Universal Robots URScript: azat_poduction_test_4.script

def azat_poduction_test_4():
  set_standard_analog_input_domain(0, 1)
  set_standard_analog_input_domain(1, 1)
  set_tool_analog_input_domain(0, 1)
  set_tool_analog_input_domain(1, 1)
  set_analog_outputdomain(0, 0)
  set_analog_outputdomain(1, 0)
  set_input_actions_to_default()
  set_target_payload(1.070000, [0.002000, 0.003000, 0.057000], [0.001723, 0.001723, 0.001723, 0.000000, 0.000000, 0.000000])
  set_tcp(p[0.0,0.0,0.0,0.0,0.0,0.0])
  set_gravity([0.0, 0.0, 9.82])
  set_tool_communication(True, 1000000, 2, 1, 1.5, 3.5)
  set_tool_output_mode(0)
  set_tool_digital_output_mode(0, 1)
  set_tool_digital_output_mode(1, 1)
  set_tool_voltage(0)
  set_safety_mode_transition_hardness(1)
  step_count_cf327c55_b5b8_495d_8ff7_12e031e14571 = 0.0
  thread Step_Counter_Thread_0ae96562_13f4_426a_a0a8_86ecd25231b4():
    while (True):
      step_count_cf327c55_b5b8_495d_8ff7_12e031e14571 = step_count_cf327c55_b5b8_495d_8ff7_12e031e14571 + 1.0
      sync()
    end
  end
  run Step_Counter_Thread_0ae96562_13f4_426a_a0a8_86ecd25231b4()
  global Plane_1=p[-0.700006141123905,1.3454883874109249E-6,0.3910559577028425,-1.2089868272251132,-1.2089999932245832,1.20858562628424]
  global Plane_2=p[0.0,0.0,0.0,0.0,0.0,0.0]
  global Point_1=p[0.6913645118948067,-0.12399382748223003,0.49223711947071,-1.2983729986843258,1.1259514972191385,-1.2203503861141718]
  $ 1 "Robot Program"
  $ 2 "Script: production_test_5.script"
  def Machining3():
    # Default parameters:
    global speed_ms = 0.3
    global speed_rads = 0.75
    global accel_mss = 3
    global accel_radss = 1.2
    global blend_radius_m = 0.001

    # Add subprograms here
    # Start of main program
    # Program generated by RoboDK v5.6.5 for UR10e on 16/10/2023 17:55:05
    # Using nominal kinematics.
    blend_radius_m = 0.001
    speed_ms = 1.000
    # set_reference(p[0.335000, -0.154000, 0.001500, 0.000000, 0.000000, 0.000000])
    set_tcp(p[0.000000, 0.000000, 0.252000, 0.000000, 0.000000, 0.000000])
    # Show Tool
    movej([0.158378, -1.225661, -2.546529, -0.940199, 1.570796, 1.729175],accel_radss,speed_rads,0,blend_radius_m)
    movel([0.158378, -1.324681, -2.603660, -0.784048, 1.570796, 1.729175],accel_mss,speed_ms,0,blend_radius_m)
    speed_ms = 0.003
    movel([0.158378, -1.328123, -2.605263, -0.779003, 1.570796, 1.729175],accel_mss,speed_ms,0,blend_radius_m)
    speed_ms = 0.008
    movel([0.158066, -1.328151, -2.605245, -0.778993, 1.570796, 1.728862],accel_mss,speed_ms,0,blend_radius_m)
    movel([0.148692, -1.330567, -2.603711, -0.778111, 1.570796, 1.719488],accel_mss,speed_ms,0,blend_radius_m)
    movel([0.142279, -1.332287, -2.602614, -0.777487, 1.570796, 1.713075],accel_mss,speed_ms,0,blend_radius_m)
    movel([0.124181, -1.337335, -2.599372, -0.775682, 1.570796, 1.694978],accel_mss,speed_ms,0,blend_radius_m)
    movel([0.122324, -1.350586, -2.590695, -0.771108, 1.570796, 1.693120],accel_mss,speed_ms,0,blend_radius_m)
    movel([0.141482, -1.345516, -2.594044, -0.772829, 1.570796, 1.712278],accel_mss,speed_ms,0,blend_radius_m)
    movel([0.146219, -1.344289, -2.594849, -0.773252, 1.570796, 1.717015],accel_mss,speed_ms,0,blend_radius_m)
    movel([0.150355, -1.343216, -2.595551, -0.773622, 1.570796, 1.721151],accel_mss,speed_ms,0,blend_radius_m)
    movel([0.155200, -1.341960, -2.596371, -0.774058, 1.570796, 1.725997],accel_mss,speed_ms,0,blend_radius_m)
    movel([0.155579, -1.341827, -2.596458, -0.774104, 1.570796, 1.726375],accel_mss,speed_ms,0,blend_radius_m)
    movel([0.156402, -1.341455, -2.596700, -0.774234, 1.570796, 1.727198],accel_mss,speed_ms,0,blend_radius_m)
    movel([0.157734, -1.333883, -2.601593, -0.776913, 1.570796, 1.728530],accel_mss,speed_ms,0,blend_radius_m)
    movel([0.158255, -1.330765, -2.603585, -0.778039, 1.570796, 1.729051],accel_mss,speed_ms,0,blend_radius_m)
    movel([0.158428, -1.329461, -2.604415, -0.778513, 1.570796, 1.729225],accel_mss,speed_ms,0,blend_radius_m)
    movel([0.158542, -1.328310, -2.605144, -0.778934, 1.570796, 1.729338],accel_mss,speed_ms,0,blend_radius_m)
    movel([0.158378, -1.328123, -2.605263, -0.779003, 1.570796, 1.729175],accel_mss,speed_ms,0,blend_radius_m)
    movel([0.158378, -1.331019, -2.606596, -0.774774, 1.570796, 1.729175],accel_mss,speed_ms,0,blend_radius_m)
    movel([0.158066, -1.331047, -2.606578, -0.774764, 1.570796, 1.728862],accel_mss,speed_ms,0,blend_radius_m)
    movel([0.148692, -1.333459, -2.605040, -0.773890, 1.570796, 1.719488],accel_mss,speed_ms,0,blend_radius_m)
    movel([0.142279, -1.335175, -2.603941, -0.773273, 1.570796, 1.713075],accel_mss,speed_ms,0,blend_radius_m)
    movel([0.124181, -1.340212, -2.600692, -0.771485, 1.570796, 1.694978],accel_mss,speed_ms,0,blend_radius_m)
    movel([0.122324, -1.353435, -2.591996, -0.766958, 1.570796, 1.693120],accel_mss,speed_ms,0,blend_radius_m)
    movel([0.141482, -1.348376, -2.595352, -0.768662, 1.570796, 1.712278],accel_mss,speed_ms,0,blend_radius_m)
    movel([0.146219, -1.347151, -2.596159, -0.769079, 1.570796, 1.717015],accel_mss,speed_ms,0,blend_radius_m)
    movel([0.150355, -1.346080, -2.596862, -0.769446, 1.570796, 1.721151],accel_mss,speed_ms,0,blend_radius_m)
    movel([0.155200, -1.344828, -2.597684, -0.769877, 1.570796, 1.725997],accel_mss,speed_ms,0,blend_radius_m)
    movel([0.155579, -1.344695, -2.597771, -0.769923, 1.570796, 1.726375],accel_mss,speed_ms,0,blend_radius_m)
    movel([0.156402, -1.344323, -2.598014, -0.770052, 1.570796, 1.727198],accel_mss,speed_ms,0,blend_radius_m)
    movel([0.157734, -1.336767, -2.602918, -0.772704, 1.570796, 1.728530],accel_mss,speed_ms,0,blend_radius_m)
    movel([0.158255, -1.333656, -2.604914, -0.773819, 1.570796, 1.729051],accel_mss,speed_ms,0,blend_radius_m)
    movel([0.158428, -1.332355, -2.605745, -0.774289, 1.570796, 1.729225],accel_mss,speed_ms,0,blend_radius_m)
    movel([0.158542, -1.331206, -2.606477, -0.774706, 1.570796, 1.729338],accel_mss,speed_ms,0,blend_radius_m)
    movel([0.158378, -1.331019, -2.606596, -0.774774, 1.570796, 1.729175],accel_mss,speed_ms,0,blend_radius_m)
    movel([0.158378, -1.297475, -2.590216, -0.824698, 1.570796, 1.729175],accel_mss,speed_ms,0,blend_radius_m)
    speed_ms = 1.000
    movel([0.162574, -1.288370, -2.595680, -0.828339, 1.570796, 1.733371],accel_mss,speed_ms,0,blend_radius_m)
    speed_ms = 0.008
    movel([0.162574, -1.315726, -2.609249, -0.787414, 1.570796, 1.733371],accel_mss,speed_ms,0,blend_radius_m)
    speed_ms = 0.003
    movel([0.162574, -1.319190, -2.610867, -0.782332, 1.570796, 1.733371],accel_mss,speed_ms,0,blend_radius_m)
    speed_ms = 0.008
    movel([0.162335, -1.318913, -2.611039, -0.782437, 1.570796, 1.733131],accel_mss,speed_ms,0,blend_radius_m)
    movel([0.162119, -1.318754, -2.611137, -0.782498, 1.570796, 1.732915],accel_mss,speed_ms,0,blend_radius_m)
    movel([0.161882, -1.318615, -2.611224, -0.782550, 1.570796, 1.732678],accel_mss,speed_ms,0,blend_radius_m)
    movel([0.161671, -1.318515, -2.611286, -0.782588, 1.570796, 1.732467],accel_mss,speed_ms,0,blend_radius_m)
    movel([0.161471, -1.318440, -2.611332, -0.782617, 1.570796, 1.732267],accel_mss,speed_ms,0,blend_radius_m)
    movel([0.160946, -1.318313, -2.611411, -0.782665, 1.570796, 1.731743],accel_mss,speed_ms,0,blend_radius_m)
    movel([0.160659, -1.318224, -2.611466, -0.782699, 1.570796, 1.731456],accel_mss,speed_ms,0,blend_radius_m)
    movel([0.160450, -1.318074, -2.611560, -0.782756, 1.570796, 1.731246],accel_mss,speed_ms,0,blend_radius_m)
    movel([0.160346, -1.317710, -2.611784, -0.782894, 1.570796, 1.731143],accel_mss,speed_ms,0,blend_radius_m)
    movel([0.160380, -1.317323, -2.612024, -0.783042, 1.570796, 1.731176],accel_mss,speed_ms,0,blend_radius_m)
    movel([0.160495, -1.316538, -2.612510, -0.783341, 1.570796, 1.731291],accel_mss,speed_ms,0,blend_radius_m)
    movel([0.160495, -1.316237, -2.612696, -0.783456, 1.570796, 1.731291],accel_mss,speed_ms,0,blend_radius_m)
    movel([0.160378, -1.316006, -2.612838, -0.783545, 1.570796, 1.731174],accel_mss,speed_ms,0,blend_radius_m)
    movel([0.160134, -1.315984, -2.612852, -0.783553, 1.570796, 1.730930],accel_mss,speed_ms,0,blend_radius_m)
    movel([0.159860, -1.316176, -2.612733, -0.783480, 1.570796, 1.730656],accel_mss,speed_ms,0,blend_radius_m)
    movel([0.159659, -1.316518, -2.612522, -0.783349, 1.570796, 1.730455],accel_mss,speed_ms,0,blend_radius_m)
    movel([0.159542, -1.316914, -2.612278, -0.783198, 1.570796, 1.730339],accel_mss,speed_ms,0,blend_radius_m)
    movel([0.159376, -1.317735, -2.611769, -0.782885, 1.570796, 1.730172],accel_mss,speed_ms,0,blend_radius_m)
    movel([0.159287, -1.318121, -2.611530, -0.782738, 1.570796, 1.730084],accel_mss,speed_ms,0,blend_radius_m)
    movel([0.159193, -1.318381, -2.611369, -0.782639, 1.570796, 1.729989],accel_mss,speed_ms,0,blend_radius_m)
    movel([0.158977, -1.318693, -2.611175, -0.782521, 1.570796, 1.729773],accel_mss,speed_ms,0,blend_radius_m)
    movel([0.158624, -1.318877, -2.611061, -0.782451, 1.570796, 1.729420],accel_mss,speed_ms,0,blend_radius_m)
    movel([0.158228, -1.319117, -2.610912, -0.782360, 1.570796, 1.729024],accel_mss,speed_ms,0,blend_radius_m)
    movel([0.157857, -1.319400, -2.610736, -0.782253, 1.570796, 1.728653],accel_mss,speed_ms,0,blend_radius_m)
    movel([0.157491, -1.319715, -2.610541, -0.782134, 1.570796, 1.728288],accel_mss,speed_ms,0,blend_radius_m)
    movel([0.157078, -1.320110, -2.610294, -0.781984, 1.570796, 1.727875],accel_mss,speed_ms,0,blend_radius_m)
    movel([0.156693, -1.320526, -2.610035, -0.781828, 1.570796, 1.727489],accel_mss,speed_ms,0,blend_radius_m)
    movel([0.156421, -1.320857, -2.609829, -0.781703, 1.570796, 1.727218],accel_mss,speed_ms,0,blend_radius_m)
    movel([0.156220, -1.321169, -2.609634, -0.781585, 1.570796, 1.727016],accel_mss,speed_ms,0,blend_radius_m)
    movel([0.156088, -1.321431, -2.609471, -0.781487, 1.570796, 1.726884],accel_mss,speed_ms,0,blend_radius_m)
    movel([0.155989, -1.321691, -2.609309, -0.781390, 1.570796, 1.726785],accel_mss,speed_ms,0,blend_radius_m)
    movel([0.155886, -1.322078, -2.609067, -0.781244, 1.570796, 1.726682],accel_mss,speed_ms,0,blend_radius_m)
    movel([0.155804, -1.322477, -2.608817, -0.781095, 1.570796, 1.726600],accel_mss,speed_ms,0,blend_radius_m)
    movel([0.155743, -1.322882, -2.608563, -0.780943, 1.570796, 1.726540],accel_mss,speed_ms,0,blend_radius_m)
    movel([0.155711, -1.323271, -2.608320, -0.780798, 1.570796, 1.726508],accel_mss,speed_ms,0,blend_radius_m)
    movel([0.155722, -1.323501, -2.608176, -0.780712, 1.570796, 1.726518],accel_mss,speed_ms,0,blend_radius_m)
    movel([0.155763, -1.323714, -2.608042, -0.780633, 1.570796, 1.726560],accel_mss,speed_ms,0,blend_radius_m)
    movel([0.155867, -1.323948, -2.607895, -0.780546, 1.570796, 1.726664],accel_mss,speed_ms,0,blend_radius_m)
    movel([0.156031, -1.324157, -2.607764, -0.780468, 1.570796, 1.726827],accel_mss,speed_ms,0,blend_radius_m)
    movel([0.156304, -1.324405, -2.607608, -0.780376, 1.570796, 1.727100],accel_mss,speed_ms,0,blend_radius_m)
    movel([0.156613, -1.324619, -2.607474, -0.780296, 1.570796, 1.727410],accel_mss,speed_ms,0,blend_radius_m)
    movel([0.156897, -1.324765, -2.607382, -0.780242, 1.570796, 1.727693],accel_mss,speed_ms,0,blend_radius_m)
    movel([0.157199, -1.324874, -2.607314, -0.780202, 1.570796, 1.727995],accel_mss,speed_ms,0,blend_radius_m)
    movel([0.157457, -1.324930, -2.607278, -0.780181, 1.570796, 1.728254],accel_mss,speed_ms,0,blend_radius_m)
    movel([0.157789, -1.324899, -2.607298, -0.780192, 1.570796, 1.728585],accel_mss,speed_ms,0,blend_radius_m)
    movel([0.157974, -1.325070, -2.607190, -0.780129, 1.570796, 1.728770],accel_mss,speed_ms,0,blend_radius_m)
    movel([0.158001, -1.325401, -2.606982, -0.780006, 1.570796, 1.728798],accel_mss,speed_ms,0,blend_radius_m)
    movel([0.157952, -1.325794, -2.606734, -0.779861, 1.570796, 1.728748],accel_mss,speed_ms,0,blend_radius_m)
    movel([0.157831, -1.326555, -2.606254, -0.779580, 1.570796, 1.728627],accel_mss,speed_ms,0,blend_radius_m)
    movel([0.157799, -1.326893, -2.606041, -0.779455, 1.570796, 1.728595],accel_mss,speed_ms,0,blend_radius_m)
    movel([0.157855, -1.327134, -2.605889, -0.779366, 1.570796, 1.728651],accel_mss,speed_ms,0,blend_radius_m)
    movel([0.158126, -1.327223, -2.605832, -0.779333, 1.570796, 1.728923],accel_mss,speed_ms,0,blend_radius_m)
    movel([0.158515, -1.327123, -2.605896, -0.779370, 1.570796, 1.729311],accel_mss,speed_ms,0,blend_radius_m)
    movel([0.158817, -1.326911, -2.606030, -0.779448, 1.570796, 1.729614],accel_mss,speed_ms,0,blend_radius_m)
    movel([0.158967, -1.326652, -2.606193, -0.779544, 1.570796, 1.729763],accel_mss,speed_ms,0,blend_radius_m)
    movel([0.159238, -1.325438, -2.606959, -0.779993, 1.570796, 1.730035],accel_mss,speed_ms,0,blend_radius_m)
    movel([0.159346, -1.325001, -2.607234, -0.780154, 1.570796, 1.730143],accel_mss,speed_ms,0,blend_radius_m)
    movel([0.159523, -1.324631, -2.607466, -0.780292, 1.570796, 1.730320],accel_mss,speed_ms,0,blend_radius_m)
    movel([0.159843, -1.324297, -2.607676, -0.780416, 1.570796, 1.730640],accel_mss,speed_ms,0,blend_radius_m)
    movel([0.160113, -1.324104, -2.607797, -0.780487, 1.570796, 1.730909],accel_mss,speed_ms,0,blend_radius_m)
    movel([0.160523, -1.323848, -2.607958, -0.780583, 1.570796, 1.731320],accel_mss,speed_ms,0,blend_radius_m)
    movel([0.161031, -1.323475, -2.608192, -0.780722, 1.570796, 1.731827],accel_mss,speed_ms,0,blend_radius_m)
    movel([0.161287, -1.323244, -2.608337, -0.780808, 1.570796, 1.732084],accel_mss,speed_ms,0,blend_radius_m)
    movel([0.161561, -1.322963, -2.608513, -0.780913, 1.570796, 1.732357],accel_mss,speed_ms,0,blend_radius_m)
    movel([0.161831, -1.322642, -2.608714, -0.781033, 1.570796, 1.732628],accel_mss,speed_ms,0,blend_radius_m)
    movel([0.162070, -1.322314, -2.608919, -0.781156, 1.570796, 1.732867],accel_mss,speed_ms,0,blend_radius_m)
    movel([0.162281, -1.321976, -2.609131, -0.781283, 1.570796, 1.733077],accel_mss,speed_ms,0,blend_radius_m)
    movel([0.162481, -1.321587, -2.609373, -0.781428, 1.570796, 1.733277],accel_mss,speed_ms,0,blend_radius_m)
    movel([0.162638, -1.321193, -2.609619, -0.781576, 1.570796, 1.733434],accel_mss,speed_ms,0,blend_radius_m)
    movel([0.162748, -1.320809, -2.609859, -0.781721, 1.570796, 1.733545],accel_mss,speed_ms,0,blend_radius_m)
    movel([0.162812, -1.320429, -2.610096, -0.781864, 1.570796, 1.733608],accel_mss,speed_ms,0,blend_radius_m)
    movel([0.162827, -1.320082, -2.610312, -0.781995, 1.570796, 1.733623],accel_mss,speed_ms,0,blend_radius_m)
    movel([0.162792, -1.319758, -2.610514, -0.782118, 1.570796, 1.733588],accel_mss,speed_ms,0,blend_radius_m)
    movel([0.162706, -1.319460, -2.610699, -0.782230, 1.570796, 1.733502],accel_mss,speed_ms,0,blend_radius_m)
    movel([0.162574, -1.319190, -2.610867, -0.782332, 1.570796, 1.733371],accel_mss,speed_ms,0,blend_radius_m)
    movel([0.162574, -1.322104, -2.612212, -0.778073, 1.570796, 1.733371],accel_mss,speed_ms,0,blend_radius_m)
    movel([0.162335, -1.321828, -2.612385, -0.778177, 1.570796, 1.733131],accel_mss,speed_ms,0,blend_radius_m)
    movel([0.162119, -1.321670, -2.612483, -0.778236, 1.570796, 1.732915],accel_mss,speed_ms,0,blend_radius_m)
    movel([0.161882, -1.321531, -2.612570, -0.778289, 1.570796, 1.732678],accel_mss,speed_ms,0,blend_radius_m)
    movel([0.161671, -1.321431, -2.612632, -0.778326, 1.570796, 1.732467],accel_mss,speed_ms,0,blend_radius_m)
    movel([0.161471, -1.321356, -2.612679, -0.778354, 1.570796, 1.732267],accel_mss,speed_ms,0,blend_radius_m)
    movel([0.160946, -1.321230, -2.612757, -0.778402, 1.570796, 1.731743],accel_mss,speed_ms,0,blend_radius_m)
    movel([0.160659, -1.321141, -2.612813, -0.778436, 1.570796, 1.731456],accel_mss,speed_ms,0,blend_radius_m)
    movel([0.160450, -1.320990, -2.612906, -0.778492, 1.570796, 1.731246],accel_mss,speed_ms,0,blend_radius_m)
    movel([0.160346, -1.320628, -2.613132, -0.778629, 1.570796, 1.731143],accel_mss,speed_ms,0,blend_radius_m)
    movel([0.160380, -1.320241, -2.613372, -0.778775, 1.570796, 1.731176],accel_mss,speed_ms,0,blend_radius_m)
    movel([0.160495, -1.319457, -2.613859, -0.779072, 1.570796, 1.731291],accel_mss,speed_ms,0,blend_radius_m)
    movel([0.160495, -1.319157, -2.614045, -0.779186, 1.570796, 1.731291],accel_mss,speed_ms,0,blend_radius_m)
    movel([0.160378, -1.318927, -2.614188, -0.779274, 1.570796, 1.731174],accel_mss,speed_ms,0,blend_radius_m)
    movel([0.160134, -1.318905, -2.614201, -0.779282, 1.570796, 1.730930],accel_mss,speed_ms,0,blend_radius_m)
    movel([0.159860, -1.319097, -2.614083, -0.779209, 1.570796, 1.730656],accel_mss,speed_ms,0,blend_radius_m)
    movel([0.159659, -1.319438, -2.613871, -0.779080, 1.570796, 1.730455],accel_mss,speed_ms,0,blend_radius_m)
    movel([0.159542, -1.319833, -2.613626, -0.778930, 1.570796, 1.730339],accel_mss,speed_ms,0,blend_radius_m)
    movel([0.159376, -1.320653, -2.613116, -0.778620, 1.570796, 1.730172],accel_mss,speed_ms,0,blend_radius_m)
    movel([0.159287, -1.321037, -2.612877, -0.778475, 1.570796, 1.730084],accel_mss,speed_ms,0,blend_radius_m)
    movel([0.159193, -1.321297, -2.612716, -0.778377, 1.570796, 1.729989],accel_mss,speed_ms,0,blend_radius_m)
    movel([0.158977, -1.321608, -2.612521, -0.778259, 1.570796, 1.729773],accel_mss,speed_ms,0,blend_radius_m)
    movel([0.158624, -1.321792, -2.612407, -0.778190, 1.570796, 1.729420],accel_mss,speed_ms,0,blend_radius_m)
    movel([0.158228, -1.322031, -2.612258, -0.778100, 1.570796, 1.729024],accel_mss,speed_ms,0,blend_radius_m)
    movel([0.157857, -1.322314, -2.612081, -0.777994, 1.570796, 1.728653],accel_mss,speed_ms,0,blend_radius_m)
    movel([0.157491, -1.322628, -2.611885, -0.777876, 1.570796, 1.728288],accel_mss,speed_ms,0,blend_radius_m)
    movel([0.157078, -1.323023, -2.611638, -0.777728, 1.570796, 1.727875],accel_mss,speed_ms,0,blend_radius_m)
    movel([0.156693, -1.323438, -2.611379, -0.777572, 1.570796, 1.727489],accel_mss,speed_ms,0,blend_radius_m)
    movel([0.156421, -1.323768, -2.611172, -0.777449, 1.570796, 1.727218],accel_mss,speed_ms,0,blend_radius_m)
    movel([0.156220, -1.324080, -2.610977, -0.777332, 1.570796, 1.727016],accel_mss,speed_ms,0,blend_radius_m)
    movel([0.156088, -1.324341, -2.610813, -0.777235, 1.570796, 1.726884],accel_mss,speed_ms,0,blend_radius_m)
    movel([0.155989, -1.324600, -2.610650, -0.777138, 1.570796, 1.726785],accel_mss,speed_ms,0,blend_radius_m)
    movel([0.155886, -1.324986, -2.610408, -0.776994, 1.570796, 1.726682],accel_mss,speed_ms,0,blend_radius_m)
    movel([0.155804, -1.325385, -2.610158, -0.776846, 1.570796, 1.726600],accel_mss,speed_ms,0,blend_radius_m)
    movel([0.155743, -1.325789, -2.609903, -0.776696, 1.570796, 1.726540],accel_mss,speed_ms,0,blend_radius_m)
    movel([0.155711, -1.326177, -2.609660, -0.776552, 1.570796, 1.726508],accel_mss,speed_ms,0,blend_radius_m)
    movel([0.155722, -1.326407, -2.609515, -0.776467, 1.570796, 1.726518],accel_mss,speed_ms,0,blend_radius_m)
    movel([0.155763, -1.326620, -2.609381, -0.776388, 1.570796, 1.726560],accel_mss,speed_ms,0,blend_radius_m)
    movel([0.155867, -1.326853, -2.609234, -0.776302, 1.570796, 1.726664],accel_mss,speed_ms,0,blend_radius_m)
    movel([0.156031, -1.327061, -2.609103, -0.776225, 1.570796, 1.726827],accel_mss,speed_ms,0,blend_radius_m)
    movel([0.156304, -1.327309, -2.608946, -0.776134, 1.570796, 1.727100],accel_mss,speed_ms,0,blend_radius_m)
    movel([0.156613, -1.327523, -2.608811, -0.776055, 1.570796, 1.727410],accel_mss,speed_ms,0,blend_radius_m)
    movel([0.156897, -1.327668, -2.608719, -0.776001, 1.570796, 1.727693],accel_mss,speed_ms,0,blend_radius_m)
    movel([0.157199, -1.327777, -2.608651, -0.775961, 1.570796, 1.727995],accel_mss,speed_ms,0,blend_radius_m)
    movel([0.157457, -1.327833, -2.608615, -0.775941, 1.570796, 1.728254],accel_mss,speed_ms,0,blend_radius_m)
    movel([0.157789, -1.327802, -2.608635, -0.775952, 1.570796, 1.728585],accel_mss,speed_ms,0,blend_radius_m)
    movel([0.157974, -1.327973, -2.608527, -0.775889, 1.570796, 1.728770],accel_mss,speed_ms,0,blend_radius_m)
    movel([0.158001, -1.328303, -2.608319, -0.775768, 1.570796, 1.728798],accel_mss,speed_ms,0,blend_radius_m)
    movel([0.157952, -1.328695, -2.608070, -0.775623, 1.570796, 1.728748],accel_mss,speed_ms,0,blend_radius_m)
    movel([0.157831, -1.329455, -2.607589, -0.775345, 1.570796, 1.728627],accel_mss,speed_ms,0,blend_radius_m)
    movel([0.157799, -1.329792, -2.607375, -0.775222, 1.570796, 1.728595],accel_mss,speed_ms,0,blend_radius_m)
    movel([0.157855, -1.330032, -2.607223, -0.775134, 1.570796, 1.728651],accel_mss,speed_ms,0,blend_radius_m)
    movel([0.158126, -1.330121, -2.607166, -0.775101, 1.570796, 1.728923],accel_mss,speed_ms,0,blend_radius_m)
    movel([0.158515, -1.330022, -2.607230, -0.775138, 1.570796, 1.729311],accel_mss,speed_ms,0,blend_radius_m)
    movel([0.158817, -1.329810, -2.607364, -0.775215, 1.570796, 1.729614],accel_mss,speed_ms,0,blend_radius_m)
    movel([0.158967, -1.329551, -2.607528, -0.775310, 1.570796, 1.729763],accel_mss,speed_ms,0,blend_radius_m)
    movel([0.159238, -1.328339, -2.608295, -0.775754, 1.570796, 1.730035],accel_mss,speed_ms,0,blend_radius_m)
    movel([0.159346, -1.327904, -2.608571, -0.775915, 1.570796, 1.730143],accel_mss,speed_ms,0,blend_radius_m)
    movel([0.159523, -1.327535, -2.608804, -0.776051, 1.570796, 1.730320],accel_mss,speed_ms,0,blend_radius_m)
    movel([0.159843, -1.327202, -2.609014, -0.776173, 1.570796, 1.730640],accel_mss,speed_ms,0,blend_radius_m)
    movel([0.160113, -1.327009, -2.609135, -0.776245, 1.570796, 1.730909],accel_mss,speed_ms,0,blend_radius_m)
    movel([0.160523, -1.326753, -2.609297, -0.776339, 1.570796, 1.731320],accel_mss,speed_ms,0,blend_radius_m)
    movel([0.161031, -1.326381, -2.609531, -0.776477, 1.570796, 1.731827],accel_mss,speed_ms,0,blend_radius_m)
    movel([0.161287, -1.326150, -2.609676, -0.776562, 1.570796, 1.732084],accel_mss,speed_ms,0,blend_radius_m)
    movel([0.161561, -1.325870, -2.609853, -0.776666, 1.570796, 1.732357],accel_mss,speed_ms,0,blend_radius_m)
    movel([0.161831, -1.325549, -2.610054, -0.776785, 1.570796, 1.732628],accel_mss,speed_ms,0,blend_radius_m)
    movel([0.162070, -1.325223, -2.610260, -0.776907, 1.570796, 1.732867],accel_mss,speed_ms,0,blend_radius_m)
    movel([0.162281, -1.324885, -2.610472, -0.777032, 1.570796, 1.733077],accel_mss,speed_ms,0,blend_radius_m)
    movel([0.162481, -1.324497, -2.610715, -0.777177, 1.570796, 1.733277],accel_mss,speed_ms,0,blend_radius_m)
    movel([0.162638, -1.324104, -2.610962, -0.777324, 1.570796, 1.733434],accel_mss,speed_ms,0,blend_radius_m)
    movel([0.162748, -1.323720, -2.611202, -0.777467, 1.570796, 1.733545],accel_mss,speed_ms,0,blend_radius_m)
    movel([0.162812, -1.323341, -2.611439, -0.777609, 1.570796, 1.733608],accel_mss,speed_ms,0,blend_radius_m)
    movel([0.162827, -1.322995, -2.611656, -0.777738, 1.570796, 1.733623],accel_mss,speed_ms,0,blend_radius_m)
    movel([0.162792, -1.322671, -2.611858, -0.777860, 1.570796, 1.733588],accel_mss,speed_ms,0,blend_radius_m)
    movel([0.162706, -1.322374, -2.612044, -0.777971, 1.570796, 1.733502],accel_mss,speed_ms,0,blend_radius_m)
    movel([0.162574, -1.322104, -2.612212, -0.778073, 1.570796, 1.733371],accel_mss,speed_ms,0,blend_radius_m)
    movel([0.162574, -1.288370, -2.595680, -0.828339, 1.570796, 1.733371],accel_mss,speed_ms,0,blend_radius_m)
    speed_ms = 1.000
    movel([0.151112, -1.291543, -2.593788, -0.827058, 1.570796, 1.721909],accel_mss,speed_ms,0,blend_radius_m)
    speed_ms = 0.008
    movel([0.151112, -1.318847, -2.607313, -0.786229, 1.570796, 1.721909],accel_mss,speed_ms,0,blend_radius_m)
    speed_ms = 0.003
    movel([0.151112, -1.322303, -2.608926, -0.781160, 1.570796, 1.721909],accel_mss,speed_ms,0,blend_radius_m)
    speed_ms = 0.008
    movel([0.151013, -1.322091, -2.609058, -0.781239, 1.570796, 1.721810],accel_mss,speed_ms,0,blend_radius_m)
    movel([0.150875, -1.321902, -2.609177, -0.781310, 1.570796, 1.721672],accel_mss,speed_ms,0,blend_radius_m)
    movel([0.150690, -1.321720, -2.609291, -0.781379, 1.570796, 1.721486],accel_mss,speed_ms,0,blend_radius_m)
    movel([0.150469, -1.321563, -2.609388, -0.781437, 1.570796, 1.721266],accel_mss,speed_ms,0,blend_radius_m)
    movel([0.150261, -1.321456, -2.609455, -0.781478, 1.570796, 1.721057],accel_mss,speed_ms,0,blend_radius_m)
    movel([0.150043, -1.321372, -2.609508, -0.781509, 1.570796, 1.720840],accel_mss,speed_ms,0,blend_radius_m)
    movel([0.149464, -1.321243, -2.609588, -0.781558, 1.570796, 1.720261],accel_mss,speed_ms,0,blend_radius_m)
    movel([0.149161, -1.321155, -2.609643, -0.781591, 1.570796, 1.719957],accel_mss,speed_ms,0,blend_radius_m)
    movel([0.148935, -1.320995, -2.609743, -0.781651, 1.570796, 1.719732],accel_mss,speed_ms,0,blend_radius_m)
    movel([0.148830, -1.320661, -2.609951, -0.781777, 1.570796, 1.719627],accel_mss,speed_ms,0,blend_radius_m)
    movel([0.148858, -1.320296, -2.610179, -0.781914, 1.570796, 1.719654],accel_mss,speed_ms,0,blend_radius_m)
    movel([0.148950, -1.319577, -2.610626, -0.782186, 1.570796, 1.719746],accel_mss,speed_ms,0,blend_radius_m)
    movel([0.148946, -1.319296, -2.610801, -0.782292, 1.570796, 1.719742],accel_mss,speed_ms,0,blend_radius_m)
    movel([0.148829, -1.319077, -2.610937, -0.782375, 1.570796, 1.719625],accel_mss,speed_ms,0,blend_radius_m)
    movel([0.148588, -1.319055, -2.610951, -0.782384, 1.570796, 1.719384],accel_mss,speed_ms,0,blend_radius_m)
    movel([0.148325, -1.319220, -2.610848, -0.782321, 1.570796, 1.719122],accel_mss,speed_ms,0,blend_radius_m)
    movel([0.148131, -1.319516, -2.610664, -0.782209, 1.570796, 1.718927],accel_mss,speed_ms,0,blend_radius_m)
    movel([0.148031, -1.319812, -2.610480, -0.782097, 1.570796, 1.718827],accel_mss,speed_ms,0,blend_radius_m)
    movel([0.147884, -1.320528, -2.610034, -0.781827, 1.570796, 1.718680],accel_mss,speed_ms,0,blend_radius_m)
    movel([0.147783, -1.320906, -2.609798, -0.781684, 1.570796, 1.718580],accel_mss,speed_ms,0,blend_radius_m)
    movel([0.147549, -1.321339, -2.609529, -0.781522, 1.570796, 1.718345],accel_mss,speed_ms,0,blend_radius_m)
    movel([0.147223, -1.321676, -2.609318, -0.781395, 1.570796, 1.718019],accel_mss,speed_ms,0,blend_radius_m)
    movel([0.146841, -1.321972, -2.609133, -0.781284, 1.570796, 1.717637],accel_mss,speed_ms,0,blend_radius_m)
    movel([0.146144, -1.322480, -2.608815, -0.781094, 1.570796, 1.716940],accel_mss,speed_ms,0,blend_radius_m)
    movel([0.145876, -1.322704, -2.608675, -0.781010, 1.570796, 1.716672],accel_mss,speed_ms,0,blend_radius_m)
    movel([0.145621, -1.322940, -2.608528, -0.780922, 1.570796, 1.716417],accel_mss,speed_ms,0,blend_radius_m)
    movel([0.145339, -1.323235, -2.608342, -0.780811, 1.570796, 1.716135],accel_mss,speed_ms,0,blend_radius_m)
    movel([0.145080, -1.323543, -2.608150, -0.780697, 1.570796, 1.715876],accel_mss,speed_ms,0,blend_radius_m)
    movel([0.144848, -1.323861, -2.607950, -0.780578, 1.570796, 1.715644],accel_mss,speed_ms,0,blend_radius_m)
    movel([0.144646, -1.324183, -2.607748, -0.780458, 1.570796, 1.715442],accel_mss,speed_ms,0,blend_radius_m)
    movel([0.144474, -1.324508, -2.607544, -0.780337, 1.570796, 1.715270],accel_mss,speed_ms,0,blend_radius_m)
    movel([0.144335, -1.324833, -2.607340, -0.780217, 1.570796, 1.715131],accel_mss,speed_ms,0,blend_radius_m)
    movel([0.144229, -1.325155, -2.607137, -0.780097, 1.570796, 1.715025],accel_mss,speed_ms,0,blend_radius_m)
    movel([0.144155, -1.325473, -2.606936, -0.779979, 1.570796, 1.714951],accel_mss,speed_ms,0,blend_radius_m)
    movel([0.144121, -1.325776, -2.606746, -0.779867, 1.570796, 1.714917],accel_mss,speed_ms,0,blend_radius_m)
    movel([0.144119, -1.326068, -2.606562, -0.779759, 1.570796, 1.714916],accel_mss,speed_ms,0,blend_radius_m)
    movel([0.144153, -1.326345, -2.606387, -0.779657, 1.570796, 1.714949],accel_mss,speed_ms,0,blend_radius_m)
    movel([0.144225, -1.326603, -2.606224, -0.779562, 1.570796, 1.715022],accel_mss,speed_ms,0,blend_radius_m)
    movel([0.144335, -1.326851, -2.606068, -0.779471, 1.570796, 1.715131],accel_mss,speed_ms,0,blend_radius_m)
    movel([0.144483, -1.327074, -2.605926, -0.779388, 1.570796, 1.715280],accel_mss,speed_ms,0,blend_radius_m)
    movel([0.144667, -1.327270, -2.605803, -0.779316, 1.570796, 1.715463],accel_mss,speed_ms,0,blend_radius_m)
    movel([0.144884, -1.327432, -2.605700, -0.779257, 1.570796, 1.715680],accel_mss,speed_ms,0,blend_radius_m)
    movel([0.145095, -1.327550, -2.605626, -0.779213, 1.570796, 1.715891],accel_mss,speed_ms,0,blend_radius_m)
    movel([0.145328, -1.327640, -2.605569, -0.779180, 1.570796, 1.716125],accel_mss,speed_ms,0,blend_radius_m)
    movel([0.145936, -1.327776, -2.605482, -0.779130, 1.570796, 1.716732],accel_mss,speed_ms,0,blend_radius_m)
    movel([0.146236, -1.327862, -2.605428, -0.779099, 1.570796, 1.717032],accel_mss,speed_ms,0,blend_radius_m)
    movel([0.146465, -1.328034, -2.605319, -0.779035, 1.570796, 1.717262],accel_mss,speed_ms,0,blend_radius_m)
    movel([0.146559, -1.328359, -2.605114, -0.778916, 1.570796, 1.717355],accel_mss,speed_ms,0,blend_radius_m)
    movel([0.146535, -1.328716, -2.604887, -0.778785, 1.570796, 1.717332],accel_mss,speed_ms,0,blend_radius_m)
    movel([0.146450, -1.329360, -2.604479, -0.778550, 1.570796, 1.717246],accel_mss,speed_ms,0,blend_radius_m)
    movel([0.146442, -1.329634, -2.604305, -0.778450, 1.570796, 1.717239],accel_mss,speed_ms,0,blend_radius_m)
    movel([0.146505, -1.329850, -2.604167, -0.778371, 1.570796, 1.717302],accel_mss,speed_ms,0,blend_radius_m)
    movel([0.146734, -1.329948, -2.604105, -0.778336, 1.570796, 1.717530],accel_mss,speed_ms,0,blend_radius_m)
    movel([0.147042, -1.329791, -2.604205, -0.778393, 1.570796, 1.717839],accel_mss,speed_ms,0,blend_radius_m)
    movel([0.147221, -1.329551, -2.604357, -0.778480, 1.570796, 1.718017],accel_mss,speed_ms,0,blend_radius_m)
    movel([0.147341, -1.329239, -2.604556, -0.778595, 1.570796, 1.718137],accel_mss,speed_ms,0,blend_radius_m)
    movel([0.147409, -1.328946, -2.604741, -0.778701, 1.570796, 1.718206],accel_mss,speed_ms,0,blend_radius_m)
    movel([0.147506, -1.328440, -2.605062, -0.778887, 1.570796, 1.718302],accel_mss,speed_ms,0,blend_radius_m)
    movel([0.147604, -1.328062, -2.605302, -0.779025, 1.570796, 1.718400],accel_mss,speed_ms,0,blend_radius_m)
    movel([0.147844, -1.327635, -2.605572, -0.779182, 1.570796, 1.718640],accel_mss,speed_ms,0,blend_radius_m)
    movel([0.148134, -1.327351, -2.605751, -0.779286, 1.570796, 1.718930],accel_mss,speed_ms,0,blend_radius_m)
    movel([0.148494, -1.327087, -2.605918, -0.779383, 1.570796, 1.719290],accel_mss,speed_ms,0,blend_radius_m)
    movel([0.149174, -1.326623, -2.606212, -0.779555, 1.570796, 1.719970],accel_mss,speed_ms,0,blend_radius_m)
    movel([0.149442, -1.326410, -2.606346, -0.779633, 1.570796, 1.720239],accel_mss,speed_ms,0,blend_radius_m)
    movel([0.149695, -1.326189, -2.606486, -0.779715, 1.570796, 1.720491],accel_mss,speed_ms,0,blend_radius_m)
    movel([0.149972, -1.325910, -2.606661, -0.779818, 1.570796, 1.720768],accel_mss,speed_ms,0,blend_radius_m)
    movel([0.150223, -1.325623, -2.606842, -0.779924, 1.570796, 1.721019],accel_mss,speed_ms,0,blend_radius_m)
    movel([0.150448, -1.325324, -2.607031, -0.780035, 1.570796, 1.721244],accel_mss,speed_ms,0,blend_radius_m)
    movel([0.150644, -1.325016, -2.607224, -0.780149, 1.570796, 1.721440],accel_mss,speed_ms,0,blend_radius_m)
    movel([0.150915, -1.324520, -2.607536, -0.780333, 1.570796, 1.721712],accel_mss,speed_ms,0,blend_radius_m)
    movel([0.151162, -1.324023, -2.607848, -0.780518, 1.570796, 1.721958],accel_mss,speed_ms,0,blend_radius_m)
    movel([0.151258, -1.323772, -2.608006, -0.780611, 1.570796, 1.722054],accel_mss,speed_ms,0,blend_radius_m)
    movel([0.151320, -1.323525, -2.608161, -0.780703, 1.570796, 1.722116],accel_mss,speed_ms,0,blend_radius_m)
    movel([0.151343, -1.323285, -2.608311, -0.780793, 1.570796, 1.722139],accel_mss,speed_ms,0,blend_radius_m)
    movel([0.151325, -1.323059, -2.608453, -0.780877, 1.570796, 1.722121],accel_mss,speed_ms,0,blend_radius_m)
    movel([0.151234, -1.322683, -2.608688, -0.781018, 1.570796, 1.722030],accel_mss,speed_ms,0,blend_radius_m)
    movel([0.151112, -1.322303, -2.608926, -0.781160, 1.570796, 1.721909],accel_mss,speed_ms,0,blend_radius_m)
    movel([0.151112, -1.325211, -2.610267, -0.776911, 1.570796, 1.721909],accel_mss,speed_ms,0,blend_radius_m)
    movel([0.151013, -1.325000, -2.610399, -0.776989, 1.570796, 1.721810],accel_mss,speed_ms,0,blend_radius_m)
    movel([0.150875, -1.324811, -2.610518, -0.777060, 1.570796, 1.721672],accel_mss,speed_ms,0,blend_radius_m)
    movel([0.150690, -1.324629, -2.610632, -0.777128, 1.570796, 1.721486],accel_mss,speed_ms,0,blend_radius_m)
    movel([0.150469, -1.324473, -2.610730, -0.777186, 1.570796, 1.721266],accel_mss,speed_ms,0,blend_radius_m)
    movel([0.150261, -1.324366, -2.610797, -0.777226, 1.570796, 1.721057],accel_mss,speed_ms,0,blend_radius_m)
    movel([0.150043, -1.324282, -2.610850, -0.777257, 1.570796, 1.720840],accel_mss,speed_ms,0,blend_radius_m)
    movel([0.149464, -1.324153, -2.610931, -0.777305, 1.570796, 1.720261],accel_mss,speed_ms,0,blend_radius_m)
    movel([0.149161, -1.324065, -2.610986, -0.777338, 1.570796, 1.719957],accel_mss,speed_ms,0,blend_radius_m)
    movel([0.148935, -1.323906, -2.611086, -0.777397, 1.570796, 1.719732],accel_mss,speed_ms,0,blend_radius_m)
    movel([0.148830, -1.323573, -2.611294, -0.777522, 1.570796, 1.719627],accel_mss,speed_ms,0,blend_radius_m)
    movel([0.148858, -1.323208, -2.611523, -0.777658, 1.570796, 1.719654],accel_mss,speed_ms,0,blend_radius_m)
    movel([0.148950, -1.322491, -2.611971, -0.777927, 1.570796, 1.719746],accel_mss,speed_ms,0,blend_radius_m)
    movel([0.148946, -1.322210, -2.612146, -0.778033, 1.570796, 1.719742],accel_mss,speed_ms,0,blend_radius_m)
    movel([0.148829, -1.321992, -2.612282, -0.778115, 1.570796, 1.719625],accel_mss,speed_ms,0,blend_radius_m)
    movel([0.148588, -1.321969, -2.612296, -0.778123, 1.570796, 1.719384],accel_mss,speed_ms,0,blend_radius_m)
    movel([0.148325, -1.322134, -2.612193, -0.778061, 1.570796, 1.719122],accel_mss,speed_ms,0,blend_radius_m)
    movel([0.148131, -1.322430, -2.612009, -0.777950, 1.570796, 1.718927],accel_mss,speed_ms,0,blend_radius_m)
    movel([0.148031, -1.322725, -2.611825, -0.777840, 1.570796, 1.718827],accel_mss,speed_ms,0,blend_radius_m)
    movel([0.147884, -1.323440, -2.611377, -0.777572, 1.570796, 1.718680],accel_mss,speed_ms,0,blend_radius_m)
    movel([0.147783, -1.323818, -2.611141, -0.777430, 1.570796, 1.718580],accel_mss,speed_ms,0,blend_radius_m)
    movel([0.147549, -1.324249, -2.610871, -0.777269, 1.570796, 1.718345],accel_mss,speed_ms,0,blend_radius_m)
    movel([0.147223, -1.324586, -2.610660, -0.777144, 1.570796, 1.718019],accel_mss,speed_ms,0,blend_radius_m)
    movel([0.146841, -1.324881, -2.610474, -0.777034, 1.570796, 1.717637],accel_mss,speed_ms,0,blend_radius_m)
    movel([0.146144, -1.325388, -2.610156, -0.776845, 1.570796, 1.716940],accel_mss,speed_ms,0,blend_radius_m)
    movel([0.145876, -1.325611, -2.610016, -0.776762, 1.570796, 1.716672],accel_mss,speed_ms,0,blend_radius_m)
    movel([0.145621, -1.325846, -2.609868, -0.776675, 1.570796, 1.716417],accel_mss,speed_ms,0,blend_radius_m)
    movel([0.145339, -1.326142, -2.609682, -0.776566, 1.570796, 1.716135],accel_mss,speed_ms,0,blend_radius_m)
    movel([0.145080, -1.326448, -2.609489, -0.776452, 1.570796, 1.715876],accel_mss,speed_ms,0,blend_radius_m)
    movel([0.144848, -1.326766, -2.609288, -0.776334, 1.570796, 1.715644],accel_mss,speed_ms,0,blend_radius_m)
    movel([0.144646, -1.327087, -2.609086, -0.776216, 1.570796, 1.715442],accel_mss,speed_ms,0,blend_radius_m)
    movel([0.144474, -1.327412, -2.608881, -0.776096, 1.570796, 1.715270],accel_mss,speed_ms,0,blend_radius_m)
    movel([0.144335, -1.327736, -2.608677, -0.775976, 1.570796, 1.715131],accel_mss,speed_ms,0,blend_radius_m)
    movel([0.144229, -1.328057, -2.608474, -0.775858, 1.570796, 1.715025],accel_mss,speed_ms,0,blend_radius_m)
    movel([0.144155, -1.328375, -2.608273, -0.775741, 1.570796, 1.714951],accel_mss,speed_ms,0,blend_radius_m)
    movel([0.144121, -1.328677, -2.608081, -0.775630, 1.570796, 1.714917],accel_mss,speed_ms,0,blend_radius_m)
    movel([0.144119, -1.328968, -2.607897, -0.775523, 1.570796, 1.714916],accel_mss,speed_ms,0,blend_radius_m)
    movel([0.144153, -1.329245, -2.607722, -0.775422, 1.570796, 1.714949],accel_mss,speed_ms,0,blend_radius_m)
    movel([0.144225, -1.329503, -2.607559, -0.775328, 1.570796, 1.715022],accel_mss,speed_ms,0,blend_radius_m)
    movel([0.144335, -1.329750, -2.607402, -0.775237, 1.570796, 1.715131],accel_mss,speed_ms,0,blend_radius_m)
    movel([0.144483, -1.329973, -2.607261, -0.775156, 1.570796, 1.715280],accel_mss,speed_ms,0,blend_radius_m)
    movel([0.144667, -1.330168, -2.607136, -0.775084, 1.570796, 1.715463],accel_mss,speed_ms,0,blend_radius_m)
    movel([0.144884, -1.330330, -2.607034, -0.775025, 1.570796, 1.715680],accel_mss,speed_ms,0,blend_radius_m)
    movel([0.145095, -1.330448, -2.606959, -0.774982, 1.570796, 1.715891],accel_mss,speed_ms,0,blend_radius_m)
    movel([0.145328, -1.330537, -2.606902, -0.774950, 1.570796, 1.716125],accel_mss,speed_ms,0,blend_radius_m)
    movel([0.145936, -1.330674, -2.606816, -0.774900, 1.570796, 1.716732],accel_mss,speed_ms,0,blend_radius_m)
    movel([0.146236, -1.330759, -2.606761, -0.774869, 1.570796, 1.717032],accel_mss,speed_ms,0,blend_radius_m)
    movel([0.146465, -1.330931, -2.606652, -0.774806, 1.570796, 1.717262],accel_mss,speed_ms,0,blend_radius_m)
    movel([0.146559, -1.331255, -2.606446, -0.774688, 1.570796, 1.717355],accel_mss,speed_ms,0,blend_radius_m)
    movel([0.146535, -1.331612, -2.606219, -0.774559, 1.570796, 1.717332],accel_mss,speed_ms,0,blend_radius_m)
    movel([0.146450, -1.332254, -2.605809, -0.774326, 1.570796, 1.717246],accel_mss,speed_ms,0,blend_radius_m)
    movel([0.146442, -1.332527, -2.605635, -0.774227, 1.570796, 1.717239],accel_mss,speed_ms,0,blend_radius_m)
    movel([0.146505, -1.332743, -2.605497, -0.774149, 1.570796, 1.717302],accel_mss,speed_ms,0,blend_radius_m)
    movel([0.146734, -1.332840, -2.605435, -0.774113, 1.570796, 1.717530],accel_mss,speed_ms,0,blend_radius_m)
    movel([0.147042, -1.332684, -2.605535, -0.774170, 1.570796, 1.717839],accel_mss,speed_ms,0,blend_radius_m)
    movel([0.147221, -1.332445, -2.605688, -0.774256, 1.570796, 1.718017],accel_mss,speed_ms,0,blend_radius_m)
    movel([0.147341, -1.332133, -2.605887, -0.774370, 1.570796, 1.718137],accel_mss,speed_ms,0,blend_radius_m)
    movel([0.147409, -1.331841, -2.606073, -0.774475, 1.570796, 1.718206],accel_mss,speed_ms,0,blend_radius_m)
    movel([0.147506, -1.331336, -2.606394, -0.774659, 1.570796, 1.718302],accel_mss,speed_ms,0,blend_radius_m)
    movel([0.147604, -1.330959, -2.606634, -0.774796, 1.570796, 1.718400],accel_mss,speed_ms,0,blend_radius_m)
    movel([0.147844, -1.330532, -2.606905, -0.774951, 1.570796, 1.718640],accel_mss,speed_ms,0,blend_radius_m)
    movel([0.148134, -1.330249, -2.607085, -0.775055, 1.570796, 1.718930],accel_mss,speed_ms,0,blend_radius_m)
    movel([0.148494, -1.329986, -2.607252, -0.775151, 1.570796, 1.719290],accel_mss,speed_ms,0,blend_radius_m)
    movel([0.149174, -1.329522, -2.607547, -0.775320, 1.570796, 1.719970],accel_mss,speed_ms,0,blend_radius_m)
    movel([0.149442, -1.329310, -2.607681, -0.775398, 1.570796, 1.720239],accel_mss,speed_ms,0,blend_radius_m)
    movel([0.149695, -1.329089, -2.607821, -0.775479, 1.570796, 1.720491],accel_mss,speed_ms,0,blend_radius_m)
    movel([0.149972, -1.328811, -2.607997, -0.775581, 1.570796, 1.720768],accel_mss,speed_ms,0,blend_radius_m)
    movel([0.150223, -1.328524, -2.608178, -0.775686, 1.570796, 1.721019],accel_mss,speed_ms,0,blend_radius_m)
    movel([0.150448, -1.328226, -2.608367, -0.775796, 1.570796, 1.721244],accel_mss,speed_ms,0,blend_radius_m)
    movel([0.150644, -1.327919, -2.608561, -0.775909, 1.570796, 1.721440],accel_mss,speed_ms,0,blend_radius_m)
    movel([0.150915, -1.327424, -2.608874, -0.776091, 1.570796, 1.721712],accel_mss,speed_ms,0,blend_radius_m)
    movel([0.151162, -1.326928, -2.609186, -0.776274, 1.570796, 1.721958],accel_mss,speed_ms,0,blend_radius_m)
    movel([0.151258, -1.326677, -2.609345, -0.776367, 1.570796, 1.722054],accel_mss,speed_ms,0,blend_radius_m)
    movel([0.151320, -1.326430, -2.609500, -0.776459, 1.570796, 1.722116],accel_mss,speed_ms,0,blend_radius_m)
    movel([0.151343, -1.326192, -2.609650, -0.776547, 1.570796, 1.722139],accel_mss,speed_ms,0,blend_radius_m)
    movel([0.151325, -1.325966, -2.609793, -0.776631, 1.570796, 1.722121],accel_mss,speed_ms,0,blend_radius_m)
    movel([0.151234, -1.325590, -2.610029, -0.776770, 1.570796, 1.722030],accel_mss,speed_ms,0,blend_radius_m)
    movel([0.151112, -1.325211, -2.610267, -0.776911, 1.570796, 1.721909],accel_mss,speed_ms,0,blend_radius_m)
    movel([0.151112, -1.291543, -2.593788, -0.827058, 1.570796, 1.721909],accel_mss,speed_ms,0,blend_radius_m)
    speed_ms = 1.000
    movel([0.139065, -1.294272, -2.592150, -0.825967, 1.570796, 1.709862],accel_mss,speed_ms,0,blend_radius_m)
    speed_ms = 0.008
    movel([0.139065, -1.321531, -2.605638, -0.785220, 1.570796, 1.709862],accel_mss,speed_ms,0,blend_radius_m)
    speed_ms = 0.003
    movel([0.139065, -1.324981, -2.607246, -0.780162, 1.570796, 1.709862],accel_mss,speed_ms,0,blend_radius_m)
    speed_ms = 0.008
    movel([0.138740, -1.324720, -2.607410, -0.780259, 1.570796, 1.709536],accel_mss,speed_ms,0,blend_radius_m)
    movel([0.138355, -1.324498, -2.607550, -0.780341, 1.570796, 1.709151],accel_mss,speed_ms,0,blend_radius_m)
    movel([0.138007, -1.324362, -2.607635, -0.780392, 1.570796, 1.708803],accel_mss,speed_ms,0,blend_radius_m)
    movel([0.137701, -1.324328, -2.607657, -0.780404, 1.570796, 1.708498],accel_mss,speed_ms,0,blend_radius_m)
    movel([0.137493, -1.324260, -2.607699, -0.780430, 1.570796, 1.708289],accel_mss,speed_ms,0,blend_radius_m)
    movel([0.137341, -1.324040, -2.607837, -0.780511, 1.570796, 1.708137],accel_mss,speed_ms,0,blend_radius_m)
    movel([0.137309, -1.323816, -2.607978, -0.780595, 1.570796, 1.708105],accel_mss,speed_ms,0,blend_radius_m)
    movel([0.137334, -1.323474, -2.608192, -0.780722, 1.570796, 1.708130],accel_mss,speed_ms,0,blend_radius_m)
    movel([0.137438, -1.322606, -2.608737, -0.781047, 1.570796, 1.708234],accel_mss,speed_ms,0,blend_radius_m)
    movel([0.137409, -1.322376, -2.608880, -0.781133, 1.570796, 1.708206],accel_mss,speed_ms,0,blend_radius_m)
    movel([0.137226, -1.322224, -2.608976, -0.781190, 1.570796, 1.708022],accel_mss,speed_ms,0,blend_radius_m)
    movel([0.136875, -1.322266, -2.608949, -0.781174, 1.570796, 1.707671],accel_mss,speed_ms,0,blend_radius_m)
    movel([0.136562, -1.322408, -2.608860, -0.781121, 1.570796, 1.707358],accel_mss,speed_ms,0,blend_radius_m)
    movel([0.136261, -1.322787, -2.608623, -0.780979, 1.570796, 1.707058],accel_mss,speed_ms,0,blend_radius_m)
    movel([0.136183, -1.323069, -2.608447, -0.780874, 1.570796, 1.706979],accel_mss,speed_ms,0,blend_radius_m)
    movel([0.136040, -1.323850, -2.607957, -0.780582, 1.570796, 1.706836],accel_mss,speed_ms,0,blend_radius_m)
    movel([0.135954, -1.324232, -2.607717, -0.780440, 1.570796, 1.706750],accel_mss,speed_ms,0,blend_radius_m)
    movel([0.135738, -1.324690, -2.607429, -0.780270, 1.570796, 1.706535],accel_mss,speed_ms,0,blend_radius_m)
    movel([0.135464, -1.324969, -2.607254, -0.780166, 1.570796, 1.706260],accel_mss,speed_ms,0,blend_radius_m)
    movel([0.134844, -1.325380, -2.606995, -0.780014, 1.570796, 1.705640],accel_mss,speed_ms,0,blend_radius_m)
    movel([0.134584, -1.325569, -2.606876, -0.779944, 1.570796, 1.705380],accel_mss,speed_ms,0,blend_radius_m)
    movel([0.134263, -1.325835, -2.606708, -0.779845, 1.570796, 1.705060],accel_mss,speed_ms,0,blend_radius_m)
    movel([0.133963, -1.326123, -2.606527, -0.779739, 1.570796, 1.704759],accel_mss,speed_ms,0,blend_radius_m)
    movel([0.133672, -1.326450, -2.606321, -0.779618, 1.570796, 1.704468],accel_mss,speed_ms,0,blend_radius_m)
    movel([0.133408, -1.326798, -2.606101, -0.779490, 1.570796, 1.704205],accel_mss,speed_ms,0,blend_radius_m)
    movel([0.133175, -1.327164, -2.605870, -0.779355, 1.570796, 1.703972],accel_mss,speed_ms,0,blend_radius_m)
    movel([0.132982, -1.327536, -2.605635, -0.779219, 1.570796, 1.703779],accel_mss,speed_ms,0,blend_radius_m)
    movel([0.132855, -1.327841, -2.605442, -0.779106, 1.570796, 1.703652],accel_mss,speed_ms,0,blend_radius_m)
    movel([0.132760, -1.328141, -2.605251, -0.778996, 1.570796, 1.703556],accel_mss,speed_ms,0,blend_radius_m)
    movel([0.132693, -1.328434, -2.605066, -0.778889, 1.570796, 1.703489],accel_mss,speed_ms,0,blend_radius_m)
    movel([0.132654, -1.328728, -2.604880, -0.778781, 1.570796, 1.703450],accel_mss,speed_ms,0,blend_radius_m)
    movel([0.132645, -1.329008, -2.604702, -0.778679, 1.570796, 1.703441],accel_mss,speed_ms,0,blend_radius_m)
    movel([0.132668, -1.329280, -2.604529, -0.778579, 1.570796, 1.703464],accel_mss,speed_ms,0,blend_radius_m)
    movel([0.132721, -1.329534, -2.604368, -0.778487, 1.570796, 1.703517],accel_mss,speed_ms,0,blend_radius_m)
    movel([0.132804, -1.329776, -2.604215, -0.778399, 1.570796, 1.703600],accel_mss,speed_ms,0,blend_radius_m)
    movel([0.132928, -1.330012, -2.604064, -0.778312, 1.570796, 1.703724],accel_mss,speed_ms,0,blend_radius_m)
    movel([0.133082, -1.330222, -2.603931, -0.778236, 1.570796, 1.703878],accel_mss,speed_ms,0,blend_radius_m)
    movel([0.133269, -1.330405, -2.603814, -0.778169, 1.570796, 1.704066],accel_mss,speed_ms,0,blend_radius_m)
    movel([0.133484, -1.330560, -2.603716, -0.778113, 1.570796, 1.704280],accel_mss,speed_ms,0,blend_radius_m)
    movel([0.133696, -1.330669, -2.603647, -0.778074, 1.570796, 1.704492],accel_mss,speed_ms,0,blend_radius_m)
    movel([0.133928, -1.330753, -2.603593, -0.778043, 1.570796, 1.704725],accel_mss,speed_ms,0,blend_radius_m)
    movel([0.134527, -1.330879, -2.603513, -0.777997, 1.570796, 1.705323],accel_mss,speed_ms,0,blend_radius_m)
    movel([0.134820, -1.330963, -2.603459, -0.777967, 1.570796, 1.705616],accel_mss,speed_ms,0,blend_radius_m)
    movel([0.135046, -1.331124, -2.603357, -0.777908, 1.570796, 1.705842],accel_mss,speed_ms,0,blend_radius_m)
    movel([0.135148, -1.331447, -2.603150, -0.777791, 1.570796, 1.705945],accel_mss,speed_ms,0,blend_radius_m)
    movel([0.135129, -1.331804, -2.602923, -0.777662, 1.570796, 1.705926],accel_mss,speed_ms,0,blend_radius_m)
    movel([0.135050, -1.332454, -2.602508, -0.777427, 1.570796, 1.705847],accel_mss,speed_ms,0,blend_radius_m)
    movel([0.135051, -1.332729, -2.602332, -0.777328, 1.570796, 1.705848],accel_mss,speed_ms,0,blend_radius_m)
    movel([0.135125, -1.332942, -2.602196, -0.777251, 1.570796, 1.705921],accel_mss,speed_ms,0,blend_radius_m)
    movel([0.135378, -1.333017, -2.602148, -0.777224, 1.570796, 1.706175],accel_mss,speed_ms,0,blend_radius_m)
    movel([0.135679, -1.332836, -2.602264, -0.777290, 1.570796, 1.706475],accel_mss,speed_ms,0,blend_radius_m)
    movel([0.135844, -1.332583, -2.602425, -0.777381, 1.570796, 1.706640],accel_mss,speed_ms,0,blend_radius_m)
    movel([0.135958, -1.332248, -2.602639, -0.777502, 1.570796, 1.706754],accel_mss,speed_ms,0,blend_radius_m)
    movel([0.136106, -1.331448, -2.603150, -0.777791, 1.570796, 1.706902],accel_mss,speed_ms,0,blend_radius_m)
    movel([0.136190, -1.331085, -2.603382, -0.777923, 1.570796, 1.706986],accel_mss,speed_ms,0,blend_radius_m)
    movel([0.136406, -1.330649, -2.603659, -0.778081, 1.570796, 1.707202],accel_mss,speed_ms,0,blend_radius_m)
    movel([0.136735, -1.330335, -2.603859, -0.778195, 1.570796, 1.707531],accel_mss,speed_ms,0,blend_radius_m)
    movel([0.137331, -1.329950, -2.604104, -0.778335, 1.570796, 1.708127],accel_mss,speed_ms,0,blend_radius_m)
    movel([0.137668, -1.329702, -2.604262, -0.778426, 1.570796, 1.708464],accel_mss,speed_ms,0,blend_radius_m)
    movel([0.137936, -1.329475, -2.604406, -0.778508, 1.570796, 1.708732],accel_mss,speed_ms,0,blend_radius_m)
    movel([0.138189, -1.329231, -2.604560, -0.778597, 1.570796, 1.708985],accel_mss,speed_ms,0,blend_radius_m)
    movel([0.138495, -1.328892, -2.604776, -0.778721, 1.570796, 1.709292],accel_mss,speed_ms,0,blend_radius_m)
    movel([0.138776, -1.328523, -2.605010, -0.778856, 1.570796, 1.709572],accel_mss,speed_ms,0,blend_radius_m)
    movel([0.139017, -1.328147, -2.605248, -0.778994, 1.570796, 1.709813],accel_mss,speed_ms,0,blend_radius_m)
    movel([0.139219, -1.327765, -2.605490, -0.779134, 1.570796, 1.710015],accel_mss,speed_ms,0,blend_radius_m)
    movel([0.139388, -1.327352, -2.605751, -0.779286, 1.570796, 1.710184],accel_mss,speed_ms,0,blend_radius_m)
    movel([0.139506, -1.326938, -2.606013, -0.779438, 1.570796, 1.710302],accel_mss,speed_ms,0,blend_radius_m)
    movel([0.139568, -1.326539, -2.606264, -0.779585, 1.570796, 1.710365],accel_mss,speed_ms,0,blend_radius_m)
    movel([0.139577, -1.326160, -2.606504, -0.779725, 1.570796, 1.710373],accel_mss,speed_ms,0,blend_radius_m)
    movel([0.139530, -1.325814, -2.606722, -0.779853, 1.570796, 1.710326],accel_mss,speed_ms,0,blend_radius_m)
    movel([0.139429, -1.325500, -2.606920, -0.779969, 1.570796, 1.710225],accel_mss,speed_ms,0,blend_radius_m)
    movel([0.139272, -1.325220, -2.607096, -0.780073, 1.570796, 1.710068],accel_mss,speed_ms,0,blend_radius_m)
    movel([0.139065, -1.324981, -2.607246, -0.780162, 1.570796, 1.709862],accel_mss,speed_ms,0,blend_radius_m)
    movel([0.139065, -1.327884, -2.608583, -0.775922, 1.570796, 1.709862],accel_mss,speed_ms,0,blend_radius_m)
    movel([0.138740, -1.327623, -2.608748, -0.776018, 1.570796, 1.709536],accel_mss,speed_ms,0,blend_radius_m)
    movel([0.138355, -1.327402, -2.608888, -0.776100, 1.570796, 1.709151],accel_mss,speed_ms,0,blend_radius_m)
    movel([0.138007, -1.327266, -2.608973, -0.776150, 1.570796, 1.708803],accel_mss,speed_ms,0,blend_radius_m)
    movel([0.137701, -1.327232, -2.608995, -0.776162, 1.570796, 1.708498],accel_mss,speed_ms,0,blend_radius_m)
    movel([0.137493, -1.327164, -2.609037, -0.776187, 1.570796, 1.708289],accel_mss,speed_ms,0,blend_radius_m)
    movel([0.137341, -1.326945, -2.609176, -0.776268, 1.570796, 1.708137],accel_mss,speed_ms,0,blend_radius_m)
    movel([0.137309, -1.326722, -2.609317, -0.776351, 1.570796, 1.708105],accel_mss,speed_ms,0,blend_radius_m)
    movel([0.137334, -1.326380, -2.609532, -0.776477, 1.570796, 1.708130],accel_mss,speed_ms,0,blend_radius_m)
    movel([0.137438, -1.325513, -2.610077, -0.776799, 1.570796, 1.708234],accel_mss,speed_ms,0,blend_radius_m)
    movel([0.137409, -1.325284, -2.610221, -0.776884, 1.570796, 1.708206],accel_mss,speed_ms,0,blend_radius_m)
    movel([0.137226, -1.325132, -2.610317, -0.776940, 1.570796, 1.708022],accel_mss,speed_ms,0,blend_radius_m)
    movel([0.136875, -1.325175, -2.610290, -0.776924, 1.570796, 1.707671],accel_mss,speed_ms,0,blend_radius_m)
    movel([0.136562, -1.325316, -2.610201, -0.776872, 1.570796, 1.707358],accel_mss,speed_ms,0,blend_radius_m)
    movel([0.136261, -1.325694, -2.609964, -0.776732, 1.570796, 1.707058],accel_mss,speed_ms,0,blend_radius_m)
    movel([0.136183, -1.325976, -2.609786, -0.776627, 1.570796, 1.706979],accel_mss,speed_ms,0,blend_radius_m)
    movel([0.136040, -1.326755, -2.609296, -0.776339, 1.570796, 1.706836],accel_mss,speed_ms,0,blend_radius_m)
    movel([0.135954, -1.327136, -2.609055, -0.776198, 1.570796, 1.706750],accel_mss,speed_ms,0,blend_radius_m)
    movel([0.135738, -1.327593, -2.608767, -0.776029, 1.570796, 1.706535],accel_mss,speed_ms,0,blend_radius_m)
    movel([0.135464, -1.327872, -2.608591, -0.775926, 1.570796, 1.706260],accel_mss,speed_ms,0,blend_radius_m)
    movel([0.134844, -1.328282, -2.608331, -0.775775, 1.570796, 1.705640],accel_mss,speed_ms,0,blend_radius_m)
    movel([0.134584, -1.328470, -2.608213, -0.775706, 1.570796, 1.705380],accel_mss,speed_ms,0,blend_radius_m)
    movel([0.134263, -1.328736, -2.608044, -0.775609, 1.570796, 1.705060],accel_mss,speed_ms,0,blend_radius_m)
    movel([0.133963, -1.329024, -2.607862, -0.775503, 1.570796, 1.704759],accel_mss,speed_ms,0,blend_radius_m)
    movel([0.133672, -1.329349, -2.607656, -0.775384, 1.570796, 1.704468],accel_mss,speed_ms,0,blend_radius_m)
    movel([0.133408, -1.329697, -2.607436, -0.775257, 1.570796, 1.704205],accel_mss,speed_ms,0,blend_radius_m)
    movel([0.133175, -1.330063, -2.607203, -0.775123, 1.570796, 1.703972],accel_mss,speed_ms,0,blend_radius_m)
    movel([0.132982, -1.330433, -2.606968, -0.774988, 1.570796, 1.703779],accel_mss,speed_ms,0,blend_radius_m)
    movel([0.132855, -1.330738, -2.606775, -0.774877, 1.570796, 1.703652],accel_mss,speed_ms,0,blend_radius_m)
    movel([0.132760, -1.331038, -2.606584, -0.774767, 1.570796, 1.703556],accel_mss,speed_ms,0,blend_radius_m)
    movel([0.132693, -1.331330, -2.606398, -0.774661, 1.570796, 1.703489],accel_mss,speed_ms,0,blend_radius_m)
    movel([0.132654, -1.331623, -2.606212, -0.774555, 1.570796, 1.703450],accel_mss,speed_ms,0,blend_radius_m)
    movel([0.132645, -1.331903, -2.606033, -0.774453, 1.570796, 1.703441],accel_mss,speed_ms,0,blend_radius_m)
    movel([0.132668, -1.332174, -2.605860, -0.774355, 1.570796, 1.703464],accel_mss,speed_ms,0,blend_radius_m)
    movel([0.132721, -1.332428, -2.605699, -0.774263, 1.570796, 1.703517],accel_mss,speed_ms,0,blend_radius_m)
    movel([0.132804, -1.332669, -2.605545, -0.774175, 1.570796, 1.703600],accel_mss,speed_ms,0,blend_radius_m)
    movel([0.132928, -1.332905, -2.605394, -0.774090, 1.570796, 1.703724],accel_mss,speed_ms,0,blend_radius_m)
    movel([0.133082, -1.333114, -2.605260, -0.774014, 1.570796, 1.703878],accel_mss,speed_ms,0,blend_radius_m)
    movel([0.133269, -1.333297, -2.605144, -0.773948, 1.570796, 1.704066],accel_mss,speed_ms,0,blend_radius_m)
    movel([0.133484, -1.333451, -2.605045, -0.773893, 1.570796, 1.704280],accel_mss,speed_ms,0,blend_radius_m)
    movel([0.133696, -1.333560, -2.604976, -0.773854, 1.570796, 1.704492],accel_mss,speed_ms,0,blend_radius_m)
    movel([0.133928, -1.333644, -2.604922, -0.773823, 1.570796, 1.704725],accel_mss,speed_ms,0,blend_radius_m)
    movel([0.134527, -1.333770, -2.604841, -0.773778, 1.570796, 1.705323],accel_mss,speed_ms,0,blend_radius_m)
    movel([0.134820, -1.333853, -2.604788, -0.773748, 1.570796, 1.705616],accel_mss,speed_ms,0,blend_radius_m)
    movel([0.135046, -1.334014, -2.604685, -0.773690, 1.570796, 1.705842],accel_mss,speed_ms,0,blend_radius_m)
    movel([0.135148, -1.334337, -2.604478, -0.773574, 1.570796, 1.705945],accel_mss,speed_ms,0,blend_radius_m)
    movel([0.135129, -1.334693, -2.604250, -0.773446, 1.570796, 1.705926],accel_mss,speed_ms,0,blend_radius_m)
    movel([0.135050, -1.335342, -2.603834, -0.773213, 1.570796, 1.705847],accel_mss,speed_ms,0,blend_radius_m)
    movel([0.135051, -1.335615, -2.603658, -0.773115, 1.570796, 1.705848],accel_mss,speed_ms,0,blend_radius_m)
    movel([0.135125, -1.335829, -2.603521, -0.773039, 1.570796, 1.705921],accel_mss,speed_ms,0,blend_radius_m)
    movel([0.135378, -1.335903, -2.603473, -0.773012, 1.570796, 1.706175],accel_mss,speed_ms,0,blend_radius_m)
    movel([0.135679, -1.335722, -2.603590, -0.773077, 1.570796, 1.706475],accel_mss,speed_ms,0,blend_radius_m)
    movel([0.135844, -1.335471, -2.603751, -0.773167, 1.570796, 1.706640],accel_mss,speed_ms,0,blend_radius_m)
    movel([0.135958, -1.335136, -2.603966, -0.773287, 1.570796, 1.706754],accel_mss,speed_ms,0,blend_radius_m)
    movel([0.136106, -1.334338, -2.604478, -0.773573, 1.570796, 1.706902],accel_mss,speed_ms,0,blend_radius_m)
    movel([0.136190, -1.333975, -2.604710, -0.773704, 1.570796, 1.706986],accel_mss,speed_ms,0,blend_radius_m)
    movel([0.136406, -1.333540, -2.604988, -0.773861, 1.570796, 1.707202],accel_mss,speed_ms,0,blend_radius_m)
    movel([0.136735, -1.333227, -2.605189, -0.773974, 1.570796, 1.707531],accel_mss,speed_ms,0,blend_radius_m)
    movel([0.137331, -1.332843, -2.605434, -0.774112, 1.570796, 1.708127],accel_mss,speed_ms,0,blend_radius_m)
    movel([0.137668, -1.332595, -2.605592, -0.774202, 1.570796, 1.708464],accel_mss,speed_ms,0,blend_radius_m)
    movel([0.137936, -1.332368, -2.605736, -0.774284, 1.570796, 1.708732],accel_mss,speed_ms,0,blend_radius_m)
    movel([0.138189, -1.332126, -2.605891, -0.774372, 1.570796, 1.708985],accel_mss,speed_ms,0,blend_radius_m)
    movel([0.138495, -1.331787, -2.606107, -0.774495, 1.570796, 1.709292],accel_mss,speed_ms,0,blend_radius_m)
    movel([0.138776, -1.331419, -2.606342, -0.774629, 1.570796, 1.709572],accel_mss,speed_ms,0,blend_radius_m)
    movel([0.139017, -1.331043, -2.606581, -0.774765, 1.570796, 1.709813],accel_mss,speed_ms,0,blend_radius_m)
    movel([0.139219, -1.330662, -2.606823, -0.774904, 1.570796, 1.710015],accel_mss,speed_ms,0,blend_radius_m)
    movel([0.139388, -1.330250, -2.607085, -0.775055, 1.570796, 1.710184],accel_mss,speed_ms,0,blend_radius_m)
    movel([0.139506, -1.329837, -2.607347, -0.775205, 1.570796, 1.710302],accel_mss,speed_ms,0,blend_radius_m)
    movel([0.139568, -1.329439, -2.607599, -0.775351, 1.570796, 1.710365],accel_mss,speed_ms,0,blend_radius_m)
    movel([0.139577, -1.329060, -2.607839, -0.775490, 1.570796, 1.710373],accel_mss,speed_ms,0,blend_radius_m)
    movel([0.139530, -1.328715, -2.608058, -0.775616, 1.570796, 1.710326],accel_mss,speed_ms,0,blend_radius_m)
    movel([0.139429, -1.328402, -2.608256, -0.775731, 1.570796, 1.710225],accel_mss,speed_ms,0,blend_radius_m)
    movel([0.139272, -1.328122, -2.608433, -0.775834, 1.570796, 1.710068],accel_mss,speed_ms,0,blend_radius_m)
    movel([0.139065, -1.327884, -2.608583, -0.775922, 1.570796, 1.709862],accel_mss,speed_ms,0,blend_radius_m)
    movel([0.139065, -1.294272, -2.592150, -0.825967, 1.570796, 1.709862],accel_mss,speed_ms,0,blend_radius_m)
    speed_ms = 1.000
    movel([0.127611, -1.297545, -2.590174, -0.824670, 1.570796, 1.698408],accel_mss,speed_ms,0,blend_radius_m)
    speed_ms = 0.008
    movel([0.127611, -1.324749, -2.603617, -0.784023, 1.570796, 1.698408],accel_mss,speed_ms,0,blend_radius_m)
    speed_ms = 0.003
    movel([0.127611, -1.328191, -2.605220, -0.778978, 1.570796, 1.698408],accel_mss,speed_ms,0,blend_radius_m)
    speed_ms = 0.008
    movel([0.127440, -1.328054, -2.605307, -0.779028, 1.570796, 1.698237],accel_mss,speed_ms,0,blend_radius_m)
    movel([0.127251, -1.327936, -2.605382, -0.779072, 1.570796, 1.698048],accel_mss,speed_ms,0,blend_radius_m)
    movel([0.127026, -1.327821, -2.605454, -0.779114, 1.570796, 1.697822],accel_mss,speed_ms,0,blend_radius_m)
    movel([0.126787, -1.327728, -2.605513, -0.779148, 1.570796, 1.697584],accel_mss,speed_ms,0,blend_radius_m)
    movel([0.126573, -1.327664, -2.605553, -0.779171, 1.570796, 1.697369],accel_mss,speed_ms,0,blend_radius_m)
    movel([0.125985, -1.327628, -2.605577, -0.779185, 1.570796, 1.696781],accel_mss,speed_ms,0,blend_radius_m)
    movel([0.125679, -1.327575, -2.605610, -0.779204, 1.570796, 1.696475],accel_mss,speed_ms,0,blend_radius_m)
    movel([0.125521, -1.327377, -2.605735, -0.779277, 1.570796, 1.696317],accel_mss,speed_ms,0,blend_radius_m)
    movel([0.125516, -1.326853, -2.606066, -0.779470, 1.570796, 1.696313],accel_mss,speed_ms,0,blend_radius_m)
    movel([0.125600, -1.326101, -2.606541, -0.779747, 1.570796, 1.696397],accel_mss,speed_ms,0,blend_radius_m)
    movel([0.125587, -1.325783, -2.606741, -0.779865, 1.570796, 1.696383],accel_mss,speed_ms,0,blend_radius_m)
    movel([0.125444, -1.325562, -2.606880, -0.779946, 1.570796, 1.696241],accel_mss,speed_ms,0,blend_radius_m)
    movel([0.125180, -1.325575, -2.606872, -0.779942, 1.570796, 1.695976],accel_mss,speed_ms,0,blend_radius_m)
    movel([0.124934, -1.325763, -2.606754, -0.779872, 1.570796, 1.695730],accel_mss,speed_ms,0,blend_radius_m)
    movel([0.124764, -1.326064, -2.606564, -0.779761, 1.570796, 1.695560],accel_mss,speed_ms,0,blend_radius_m)
    movel([0.124671, -1.326394, -2.606356, -0.779639, 1.570796, 1.695467],accel_mss,speed_ms,0,blend_radius_m)
    movel([0.124556, -1.327067, -2.605931, -0.779391, 1.570796, 1.695352],accel_mss,speed_ms,0,blend_radius_m)
    movel([0.124482, -1.327412, -2.605713, -0.779264, 1.570796, 1.695278],accel_mss,speed_ms,0,blend_radius_m)
    movel([0.124276, -1.327860, -2.605430, -0.779099, 1.570796, 1.695072],accel_mss,speed_ms,0,blend_radius_m)
    movel([0.124023, -1.328122, -2.605264, -0.779003, 1.570796, 1.694819],accel_mss,speed_ms,0,blend_radius_m)
    movel([0.123580, -1.328410, -2.605082, -0.778898, 1.570796, 1.694377],accel_mss,speed_ms,0,blend_radius_m)
    movel([0.123259, -1.328671, -2.604916, -0.778802, 1.570796, 1.694055],accel_mss,speed_ms,0,blend_radius_m)
    movel([0.122897, -1.329001, -2.604707, -0.778681, 1.570796, 1.693693],accel_mss,speed_ms,0,blend_radius_m)
    movel([0.122545, -1.329352, -2.604484, -0.778553, 1.570796, 1.693342],accel_mss,speed_ms,0,blend_radius_m)
    movel([0.122206, -1.329730, -2.604244, -0.778415, 1.570796, 1.693002],accel_mss,speed_ms,0,blend_radius_m)
    movel([0.121955, -1.330049, -2.604041, -0.778299, 1.570796, 1.692752],accel_mss,speed_ms,0,blend_radius_m)
    movel([0.121722, -1.330398, -2.603819, -0.778172, 1.570796, 1.692518],accel_mss,speed_ms,0,blend_radius_m)
    movel([0.121526, -1.330752, -2.603594, -0.778043, 1.570796, 1.692322],accel_mss,speed_ms,0,blend_radius_m)
    movel([0.121393, -1.331054, -2.603401, -0.777934, 1.570796, 1.692189],accel_mss,speed_ms,0,blend_radius_m)
    movel([0.121285, -1.331355, -2.603210, -0.777825, 1.570796, 1.692081],accel_mss,speed_ms,0,blend_radius_m)
    movel([0.121208, -1.331658, -2.603016, -0.777715, 1.570796, 1.692004],accel_mss,speed_ms,0,blend_radius_m)
    movel([0.121159, -1.331955, -2.602826, -0.777607, 1.570796, 1.691956],accel_mss,speed_ms,0,blend_radius_m)
    movel([0.121141, -1.332239, -2.602645, -0.777505, 1.570796, 1.691937],accel_mss,speed_ms,0,blend_radius_m)
    movel([0.121154, -1.332514, -2.602469, -0.777405, 1.570796, 1.691950],accel_mss,speed_ms,0,blend_radius_m)
    movel([0.121197, -1.332772, -2.602305, -0.777313, 1.570796, 1.691993],accel_mss,speed_ms,0,blend_radius_m)
    movel([0.121270, -1.333011, -2.602152, -0.777226, 1.570796, 1.692067],accel_mss,speed_ms,0,blend_radius_m)
    movel([0.121385, -1.333261, -2.601992, -0.777136, 1.570796, 1.692182],accel_mss,speed_ms,0,blend_radius_m)
    movel([0.121540, -1.333484, -2.601849, -0.777056, 1.570796, 1.692336],accel_mss,speed_ms,0,blend_radius_m)
    movel([0.121728, -1.333679, -2.601724, -0.776986, 1.570796, 1.692524],accel_mss,speed_ms,0,blend_radius_m)
    movel([0.121937, -1.333833, -2.601625, -0.776931, 1.570796, 1.692734],accel_mss,speed_ms,0,blend_radius_m)
    movel([0.122162, -1.333946, -2.601553, -0.776890, 1.570796, 1.692958],accel_mss,speed_ms,0,blend_radius_m)
    movel([0.122408, -1.334030, -2.601499, -0.776860, 1.570796, 1.693205],accel_mss,speed_ms,0,blend_radius_m)
    movel([0.122650, -1.334078, -2.601468, -0.776843, 1.570796, 1.693446],accel_mss,speed_ms,0,blend_radius_m)
    movel([0.122992, -1.334114, -2.601445, -0.776830, 1.570796, 1.693788],accel_mss,speed_ms,0,blend_radius_m)
    movel([0.123282, -1.334208, -2.601384, -0.776796, 1.570796, 1.694078],accel_mss,speed_ms,0,blend_radius_m)
    movel([0.123442, -1.334457, -2.601225, -0.776707, 1.570796, 1.694238],accel_mss,speed_ms,0,blend_radius_m)
    movel([0.123440, -1.335015, -2.600866, -0.776507, 1.570796, 1.694236],accel_mss,speed_ms,0,blend_radius_m)
    movel([0.123361, -1.335702, -2.600425, -0.776262, 1.570796, 1.694157],accel_mss,speed_ms,0,blend_radius_m)
    movel([0.123353, -1.335975, -2.600249, -0.776165, 1.570796, 1.694150],accel_mss,speed_ms,0,blend_radius_m)
    movel([0.123425, -1.336183, -2.600115, -0.776091, 1.570796, 1.694221],accel_mss,speed_ms,0,blend_radius_m)
    movel([0.123802, -1.336233, -2.600083, -0.776073, 1.570796, 1.694598],accel_mss,speed_ms,0,blend_radius_m)
    movel([0.124244, -1.336046, -2.600204, -0.776140, 1.570796, 1.695041],accel_mss,speed_ms,0,blend_radius_m)
    movel([0.124489, -1.335744, -2.600398, -0.776247, 1.570796, 1.695285],accel_mss,speed_ms,0,blend_radius_m)
    movel([0.124625, -1.335209, -2.600742, -0.776438, 1.570796, 1.695421],accel_mss,speed_ms,0,blend_radius_m)
    movel([0.124718, -1.334643, -2.601106, -0.776641, 1.570796, 1.695514],accel_mss,speed_ms,0,blend_radius_m)
    movel([0.124809, -1.334250, -2.601358, -0.776781, 1.570796, 1.695605],accel_mss,speed_ms,0,blend_radius_m)
    movel([0.125007, -1.333846, -2.601617, -0.776926, 1.570796, 1.695804],accel_mss,speed_ms,0,blend_radius_m)
    movel([0.125281, -1.333537, -2.601815, -0.777037, 1.570796, 1.696078],accel_mss,speed_ms,0,blend_radius_m)
    movel([0.125570, -1.333303, -2.601965, -0.777121, 1.570796, 1.696366],accel_mss,speed_ms,0,blend_radius_m)
    movel([0.126022, -1.332974, -2.602176, -0.777240, 1.570796, 1.696818],accel_mss,speed_ms,0,blend_radius_m)
    movel([0.126284, -1.332767, -2.602308, -0.777314, 1.570796, 1.697081],accel_mss,speed_ms,0,blend_radius_m)
    movel([0.126586, -1.332502, -2.602477, -0.777410, 1.570796, 1.697382],accel_mss,speed_ms,0,blend_radius_m)
    movel([0.126868, -1.332225, -2.602654, -0.777510, 1.570796, 1.697665],accel_mss,speed_ms,0,blend_radius_m)
    movel([0.127161, -1.331902, -2.602860, -0.777627, 1.570796, 1.697957],accel_mss,speed_ms,0,blend_radius_m)
    movel([0.127406, -1.331590, -2.603060, -0.777740, 1.570796, 1.698202],accel_mss,speed_ms,0,blend_radius_m)
    movel([0.127623, -1.331263, -2.603268, -0.777858, 1.570796, 1.698419],accel_mss,speed_ms,0,blend_radius_m)
    movel([0.127810, -1.330928, -2.603481, -0.777979, 1.570796, 1.698607],accel_mss,speed_ms,0,blend_radius_m)
    movel([0.127985, -1.330525, -2.603738, -0.778126, 1.570796, 1.698782],accel_mss,speed_ms,0,blend_radius_m)
    movel([0.128103, -1.330136, -2.603986, -0.778267, 1.570796, 1.698899],accel_mss,speed_ms,0,blend_radius_m)
    movel([0.128165, -1.329755, -2.604228, -0.778406, 1.570796, 1.698962],accel_mss,speed_ms,0,blend_radius_m)
    movel([0.128170, -1.329392, -2.604458, -0.778539, 1.570796, 1.698966],accel_mss,speed_ms,0,blend_radius_m)
    movel([0.128113, -1.329044, -2.604679, -0.778666, 1.570796, 1.698910],accel_mss,speed_ms,0,blend_radius_m)
    movel([0.127997, -1.328722, -2.604883, -0.778783, 1.570796, 1.698794],accel_mss,speed_ms,0,blend_radius_m)
    movel([0.127830, -1.328437, -2.605064, -0.778888, 1.570796, 1.698626],accel_mss,speed_ms,0,blend_radius_m)
    movel([0.127611, -1.328191, -2.605220, -0.778978, 1.570796, 1.698408],accel_mss,speed_ms,0,blend_radius_m)
    movel([0.127611, -1.331087, -2.606552, -0.774749, 1.570796, 1.698408],accel_mss,speed_ms,0,blend_radius_m)
    movel([0.127440, -1.330951, -2.606639, -0.774799, 1.570796, 1.698237],accel_mss,speed_ms,0,blend_radius_m)
    movel([0.127251, -1.330832, -2.606715, -0.774842, 1.570796, 1.698048],accel_mss,speed_ms,0,blend_radius_m)
    movel([0.127026, -1.330718, -2.606787, -0.774884, 1.570796, 1.697822],accel_mss,speed_ms,0,blend_radius_m)
    movel([0.126787, -1.330625, -2.606846, -0.774918, 1.570796, 1.697584],accel_mss,speed_ms,0,blend_radius_m)
    movel([0.126573, -1.330562, -2.606887, -0.774941, 1.570796, 1.697369],accel_mss,speed_ms,0,blend_radius_m)
    movel([0.125985, -1.330525, -2.606910, -0.774954, 1.570796, 1.696781],accel_mss,speed_ms,0,blend_radius_m)
    movel([0.125679, -1.330472, -2.606944, -0.774973, 1.570796, 1.696475],accel_mss,speed_ms,0,blend_radius_m)
    movel([0.125521, -1.330275, -2.607069, -0.775045, 1.570796, 1.696317],accel_mss,speed_ms,0,blend_radius_m)
    movel([0.125516, -1.329752, -2.607401, -0.775236, 1.570796, 1.696313],accel_mss,speed_ms,0,blend_radius_m)
    movel([0.125600, -1.329002, -2.607876, -0.775511, 1.570796, 1.696397],accel_mss,speed_ms,0,blend_radius_m)
    movel([0.125587, -1.328684, -2.608077, -0.775628, 1.570796, 1.696383],accel_mss,speed_ms,0,blend_radius_m)
    movel([0.125444, -1.328464, -2.608216, -0.775708, 1.570796, 1.696241],accel_mss,speed_ms,0,blend_radius_m)
    movel([0.125180, -1.328476, -2.608209, -0.775704, 1.570796, 1.695976],accel_mss,speed_ms,0,blend_radius_m)
    movel([0.124934, -1.328665, -2.608090, -0.775635, 1.570796, 1.695730],accel_mss,speed_ms,0,blend_radius_m)
    movel([0.124764, -1.328965, -2.607900, -0.775525, 1.570796, 1.695560],accel_mss,speed_ms,0,blend_radius_m)
    movel([0.124671, -1.329294, -2.607691, -0.775404, 1.570796, 1.695467],accel_mss,speed_ms,0,blend_radius_m)
    movel([0.124556, -1.329965, -2.607265, -0.775158, 1.570796, 1.695352],accel_mss,speed_ms,0,blend_radius_m)
    movel([0.124482, -1.330309, -2.607047, -0.775033, 1.570796, 1.695278],accel_mss,speed_ms,0,blend_radius_m)
    movel([0.124276, -1.330757, -2.606763, -0.774870, 1.570796, 1.695072],accel_mss,speed_ms,0,blend_radius_m)
    movel([0.124023, -1.331019, -2.606596, -0.774774, 1.570796, 1.694819],accel_mss,speed_ms,0,blend_radius_m)
    movel([0.123580, -1.331305, -2.606414, -0.774670, 1.570796, 1.694377],accel_mss,speed_ms,0,blend_radius_m)
    movel([0.123259, -1.331567, -2.606247, -0.774575, 1.570796, 1.694055],accel_mss,speed_ms,0,blend_radius_m)
    movel([0.122897, -1.331895, -2.606038, -0.774456, 1.570796, 1.693693],accel_mss,speed_ms,0,blend_radius_m)
    movel([0.122545, -1.332246, -2.605814, -0.774328, 1.570796, 1.693342],accel_mss,speed_ms,0,blend_radius_m)
    movel([0.122206, -1.332623, -2.605574, -0.774192, 1.570796, 1.693002],accel_mss,speed_ms,0,blend_radius_m)
    movel([0.121955, -1.332942, -2.605370, -0.774077, 1.570796, 1.692752],accel_mss,speed_ms,0,blend_radius_m)
    movel([0.121722, -1.333290, -2.605148, -0.773951, 1.570796, 1.692518],accel_mss,speed_ms,0,blend_radius_m)
    movel([0.121526, -1.333643, -2.604922, -0.773824, 1.570796, 1.692322],accel_mss,speed_ms,0,blend_radius_m)
    movel([0.121393, -1.333944, -2.604730, -0.773715, 1.570796, 1.692189],accel_mss,speed_ms,0,blend_radius_m)
    movel([0.121285, -1.334244, -2.604538, -0.773607, 1.570796, 1.692081],accel_mss,speed_ms,0,blend_radius_m)
    movel([0.121208, -1.334547, -2.604344, -0.773498, 1.570796, 1.692004],accel_mss,speed_ms,0,blend_radius_m)
    movel([0.121159, -1.334844, -2.604153, -0.773392, 1.570796, 1.691956],accel_mss,speed_ms,0,blend_radius_m)
    movel([0.121141, -1.335127, -2.603972, -0.773290, 1.570796, 1.691937],accel_mss,speed_ms,0,blend_radius_m)
    movel([0.121154, -1.335402, -2.603795, -0.773192, 1.570796, 1.691950],accel_mss,speed_ms,0,blend_radius_m)
    movel([0.121197, -1.335658, -2.603631, -0.773100, 1.570796, 1.691993],accel_mss,speed_ms,0,blend_radius_m)
    movel([0.121270, -1.335897, -2.603477, -0.773014, 1.570796, 1.692067],accel_mss,speed_ms,0,blend_radius_m)
    movel([0.121385, -1.336147, -2.603317, -0.772925, 1.570796, 1.692182],accel_mss,speed_ms,0,blend_radius_m)
    movel([0.121540, -1.336369, -2.603174, -0.772846, 1.570796, 1.692336],accel_mss,speed_ms,0,blend_radius_m)
    movel([0.121728, -1.336564, -2.603048, -0.772776, 1.570796, 1.692524],accel_mss,speed_ms,0,blend_radius_m)
    movel([0.121937, -1.336717, -2.602950, -0.772722, 1.570796, 1.692734],accel_mss,speed_ms,0,blend_radius_m)
    movel([0.122162, -1.336830, -2.602877, -0.772682, 1.570796, 1.692958],accel_mss,speed_ms,0,blend_radius_m)
    movel([0.122408, -1.336915, -2.602823, -0.772652, 1.570796, 1.693205],accel_mss,speed_ms,0,blend_radius_m)
    movel([0.122650, -1.336963, -2.602792, -0.772635, 1.570796, 1.693446],accel_mss,speed_ms,0,blend_radius_m)
    movel([0.122992, -1.336998, -2.602769, -0.772622, 1.570796, 1.693788],accel_mss,speed_ms,0,blend_radius_m)
    movel([0.123282, -1.337092, -2.602708, -0.772588, 1.570796, 1.694078],accel_mss,speed_ms,0,blend_radius_m)
    movel([0.123442, -1.337340, -2.602549, -0.772500, 1.570796, 1.694238],accel_mss,speed_ms,0,blend_radius_m)
    movel([0.123440, -1.337897, -2.602189, -0.772302, 1.570796, 1.694236],accel_mss,speed_ms,0,blend_radius_m)
    movel([0.123361, -1.338583, -2.601746, -0.772060, 1.570796, 1.694157],accel_mss,speed_ms,0,blend_radius_m)
    movel([0.123353, -1.338855, -2.601570, -0.771963, 1.570796, 1.694150],accel_mss,speed_ms,0,blend_radius_m)
    movel([0.123425, -1.339062, -2.601436, -0.771890, 1.570796, 1.694221],accel_mss,speed_ms,0,blend_radius_m)
    movel([0.123802, -1.339113, -2.601404, -0.771872, 1.570796, 1.694598],accel_mss,speed_ms,0,blend_radius_m)
    movel([0.124244, -1.338926, -2.601525, -0.771939, 1.570796, 1.695041],accel_mss,speed_ms,0,blend_radius_m)
    movel([0.124489, -1.338625, -2.601719, -0.772045, 1.570796, 1.695285],accel_mss,speed_ms,0,blend_radius_m)
    movel([0.124625, -1.338090, -2.602065, -0.772234, 1.570796, 1.695421],accel_mss,speed_ms,0,blend_radius_m)
    movel([0.124718, -1.337526, -2.602429, -0.772434, 1.570796, 1.695514],accel_mss,speed_ms,0,blend_radius_m)
    movel([0.124809, -1.337133, -2.602682, -0.772574, 1.570796, 1.695605],accel_mss,speed_ms,0,blend_radius_m)
    movel([0.125007, -1.336730, -2.602941, -0.772717, 1.570796, 1.695804],accel_mss,speed_ms,0,blend_radius_m)
    movel([0.125281, -1.336422, -2.603140, -0.772827, 1.570796, 1.696078],accel_mss,speed_ms,0,blend_radius_m)
    movel([0.125570, -1.336189, -2.603290, -0.772910, 1.570796, 1.696366],accel_mss,speed_ms,0,blend_radius_m)
    movel([0.126022, -1.335860, -2.603501, -0.773028, 1.570796, 1.696818],accel_mss,speed_ms,0,blend_radius_m)
    movel([0.126284, -1.335654, -2.603634, -0.773102, 1.570796, 1.697081],accel_mss,speed_ms,0,blend_radius_m)
    movel([0.126586, -1.335390, -2.603803, -0.773196, 1.570796, 1.697382],accel_mss,speed_ms,0,blend_radius_m)
    movel([0.126868, -1.335113, -2.603981, -0.773295, 1.570796, 1.697665],accel_mss,speed_ms,0,blend_radius_m)
    movel([0.127161, -1.334790, -2.604188, -0.773411, 1.570796, 1.697957],accel_mss,speed_ms,0,blend_radius_m)
    movel([0.127406, -1.334479, -2.604387, -0.773523, 1.570796, 1.698202],accel_mss,speed_ms,0,blend_radius_m)
    movel([0.127623, -1.334153, -2.604596, -0.773640, 1.570796, 1.698419],accel_mss,speed_ms,0,blend_radius_m)
    movel([0.127810, -1.333819, -2.604810, -0.773760, 1.570796, 1.698607],accel_mss,speed_ms,0,blend_radius_m)
    movel([0.127985, -1.333417, -2.605067, -0.773905, 1.570796, 1.698782],accel_mss,speed_ms,0,blend_radius_m)
    movel([0.128103, -1.333028, -2.605315, -0.774046, 1.570796, 1.698899],accel_mss,speed_ms,0,blend_radius_m)
    movel([0.128165, -1.332648, -2.605558, -0.774183, 1.570796, 1.698962],accel_mss,speed_ms,0,blend_radius_m)
    movel([0.128170, -1.332286, -2.605789, -0.774314, 1.570796, 1.698966],accel_mss,speed_ms,0,blend_radius_m)
    movel([0.128113, -1.331939, -2.606010, -0.774440, 1.570796, 1.698910],accel_mss,speed_ms,0,blend_radius_m)
    movel([0.127997, -1.331617, -2.606215, -0.774557, 1.570796, 1.698794],accel_mss,speed_ms,0,blend_radius_m)
    movel([0.127830, -1.331333, -2.606396, -0.774660, 1.570796, 1.698626],accel_mss,speed_ms,0,blend_radius_m)
    movel([0.127611, -1.331087, -2.606552, -0.774749, 1.570796, 1.698408],accel_mss,speed_ms,0,blend_radius_m)
    movel([0.127611, -1.297545, -2.590174, -0.824670, 1.570796, 1.698408],accel_mss,speed_ms,0,blend_radius_m)
    speed_ms = 1.000
    movel([0.134188, -1.285153, -2.597586, -0.829650, 1.570796, 1.704984],accel_mss,speed_ms,0,blend_radius_m)
    speed_ms = 0.008
    movel([0.134188, -1.312562, -2.611198, -0.788629, 1.570796, 1.704984],accel_mss,speed_ms,0,blend_radius_m)
    speed_ms = 0.003
    movel([0.134188, -1.316033, -2.612822, -0.783535, 1.570796, 1.704984],accel_mss,speed_ms,0,blend_radius_m)
    speed_ms = 0.008
    movel([0.133863, -1.316551, -2.612502, -0.783336, 1.570796, 1.704659],accel_mss,speed_ms,0,blend_radius_m)
    movel([0.133488, -1.317060, -2.612187, -0.783142, 1.570796, 1.704284],accel_mss,speed_ms,0,blend_radius_m)
    movel([0.133051, -1.317573, -2.611870, -0.782946, 1.570796, 1.703848],accel_mss,speed_ms,0,blend_radius_m)
    movel([0.132574, -1.318070, -2.611562, -0.782757, 1.570796, 1.703370],accel_mss,speed_ms,0,blend_radius_m)
    movel([0.132063, -1.318539, -2.611271, -0.782579, 1.570796, 1.702859],accel_mss,speed_ms,0,blend_radius_m)
    movel([0.131519, -1.318983, -2.610995, -0.782411, 1.570796, 1.702316],accel_mss,speed_ms,0,blend_radius_m)
    movel([0.130956, -1.319391, -2.610742, -0.782256, 1.570796, 1.701752],accel_mss,speed_ms,0,blend_radius_m)
    movel([0.130359, -1.319772, -2.610505, -0.782112, 1.570796, 1.701155],accel_mss,speed_ms,0,blend_radius_m)
    movel([0.129758, -1.320108, -2.610295, -0.781985, 1.570796, 1.700554],accel_mss,speed_ms,0,blend_radius_m)
    movel([0.129170, -1.320393, -2.610118, -0.781878, 1.570796, 1.699967],accel_mss,speed_ms,0,blend_radius_m)
    movel([0.128584, -1.320634, -2.609968, -0.781787, 1.570796, 1.699380],accel_mss,speed_ms,0,blend_radius_m)
    movel([0.127997, -1.320825, -2.609849, -0.781715, 1.570796, 1.698794],accel_mss,speed_ms,0,blend_radius_m)
    movel([0.127420, -1.320970, -2.609758, -0.781660, 1.570796, 1.698216],accel_mss,speed_ms,0,blend_radius_m)
    movel([0.126855, -1.321064, -2.609700, -0.781625, 1.570796, 1.697652],accel_mss,speed_ms,0,blend_radius_m)
    movel([0.126287, -1.321108, -2.609672, -0.781608, 1.570796, 1.697084],accel_mss,speed_ms,0,blend_radius_m)
    movel([0.125741, -1.321106, -2.609674, -0.781609, 1.570796, 1.696538],accel_mss,speed_ms,0,blend_radius_m)
    movel([0.125218, -1.321051, -2.609708, -0.781630, 1.570796, 1.696014],accel_mss,speed_ms,0,blend_radius_m)
    movel([0.124728, -1.320944, -2.609775, -0.781670, 1.570796, 1.695524],accel_mss,speed_ms,0,blend_radius_m)
    movel([0.124274, -1.320792, -2.609870, -0.781727, 1.570796, 1.695070],accel_mss,speed_ms,0,blend_radius_m)
    movel([0.123865, -1.320593, -2.609994, -0.781802, 1.570796, 1.694662],accel_mss,speed_ms,0,blend_radius_m)
    movel([0.123500, -1.320342, -2.610150, -0.781897, 1.570796, 1.694296],accel_mss,speed_ms,0,blend_radius_m)
    movel([0.123179, -1.320047, -2.610334, -0.782008, 1.570796, 1.693975],accel_mss,speed_ms,0,blend_radius_m)
    movel([0.122903, -1.319702, -2.610548, -0.782139, 1.570796, 1.693699],accel_mss,speed_ms,0,blend_radius_m)
    movel([0.122698, -1.319340, -2.610773, -0.782275, 1.570796, 1.693494],accel_mss,speed_ms,0,blend_radius_m)
    movel([0.122566, -1.318973, -2.611001, -0.782414, 1.570796, 1.693362],accel_mss,speed_ms,0,blend_radius_m)
    movel([0.122485, -1.318575, -2.611248, -0.782565, 1.570796, 1.693281],accel_mss,speed_ms,0,blend_radius_m)
    movel([0.122458, -1.318152, -2.611511, -0.782726, 1.570796, 1.693255],accel_mss,speed_ms,0,blend_radius_m)
    movel([0.122486, -1.317708, -2.611786, -0.782895, 1.570796, 1.693283],accel_mss,speed_ms,0,blend_radius_m)
    movel([0.122590, -1.317105, -2.612159, -0.783125, 1.570796, 1.693386],accel_mss,speed_ms,0,blend_radius_m)
    movel([0.122748, -1.316487, -2.612541, -0.783361, 1.570796, 1.693544],accel_mss,speed_ms,0,blend_radius_m)
    movel([0.122933, -1.315949, -2.612873, -0.783567, 1.570796, 1.693730],accel_mss,speed_ms,0,blend_radius_m)
    movel([0.123172, -1.315419, -2.613201, -0.783770, 1.570796, 1.693969],accel_mss,speed_ms,0,blend_radius_m)
    movel([0.123393, -1.315020, -2.613446, -0.783923, 1.570796, 1.694190],accel_mss,speed_ms,0,blend_radius_m)
    movel([0.123730, -1.314665, -2.613665, -0.784059, 1.570796, 1.694526],accel_mss,speed_ms,0,blend_radius_m)
    movel([0.124098, -1.314527, -2.613750, -0.784113, 1.570796, 1.694894],accel_mss,speed_ms,0,blend_radius_m)
    movel([0.124241, -1.314688, -2.613651, -0.784051, 1.570796, 1.695037],accel_mss,speed_ms,0,blend_radius_m)
    movel([0.124444, -1.314827, -2.613565, -0.783997, 1.570796, 1.695240],accel_mss,speed_ms,0,blend_radius_m)
    movel([0.125111, -1.314823, -2.613568, -0.783999, 1.570796, 1.695907],accel_mss,speed_ms,0,blend_radius_m)
    movel([0.125436, -1.314859, -2.613545, -0.783985, 1.570796, 1.696233],accel_mss,speed_ms,0,blend_radius_m)
    movel([0.125718, -1.314950, -2.613489, -0.783950, 1.570796, 1.696514],accel_mss,speed_ms,0,blend_radius_m)
    movel([0.126039, -1.315070, -2.613415, -0.783904, 1.570796, 1.696836],accel_mss,speed_ms,0,blend_radius_m)
    movel([0.126622, -1.315350, -2.613243, -0.783796, 1.570796, 1.697418],accel_mss,speed_ms,0,blend_radius_m)
    movel([0.127045, -1.315603, -2.613087, -0.783699, 1.570796, 1.697841],accel_mss,speed_ms,0,blend_radius_m)
    movel([0.127393, -1.315859, -2.612929, -0.783601, 1.570796, 1.698189],accel_mss,speed_ms,0,blend_radius_m)
    movel([0.127590, -1.316085, -2.612789, -0.783515, 1.570796, 1.698386],accel_mss,speed_ms,0,blend_radius_m)
    movel([0.127760, -1.316388, -2.612603, -0.783399, 1.570796, 1.698556],accel_mss,speed_ms,0,blend_radius_m)
    movel([0.127974, -1.316623, -2.612457, -0.783309, 1.570796, 1.698770],accel_mss,speed_ms,0,blend_radius_m)
    movel([0.128319, -1.316762, -2.612371, -0.783256, 1.570796, 1.699116],accel_mss,speed_ms,0,blend_radius_m)
    movel([0.128768, -1.316702, -2.612409, -0.783279, 1.570796, 1.699565],accel_mss,speed_ms,0,blend_radius_m)
    movel([0.129117, -1.316518, -2.612522, -0.783349, 1.570796, 1.699913],accel_mss,speed_ms,0,blend_radius_m)
    movel([0.129483, -1.316194, -2.612722, -0.783473, 1.570796, 1.700280],accel_mss,speed_ms,0,blend_radius_m)
    movel([0.129679, -1.315947, -2.612875, -0.783568, 1.570796, 1.700476],accel_mss,speed_ms,0,blend_radius_m)
    movel([0.129887, -1.315461, -2.613175, -0.783754, 1.570796, 1.700683],accel_mss,speed_ms,0,blend_radius_m)
    movel([0.129841, -1.315049, -2.613428, -0.783912, 1.570796, 1.700637],accel_mss,speed_ms,0,blend_radius_m)
    movel([0.129723, -1.314890, -2.613526, -0.783973, 1.570796, 1.700519],accel_mss,speed_ms,0,blend_radius_m)
    movel([0.129545, -1.314766, -2.613602, -0.784021, 1.570796, 1.700341],accel_mss,speed_ms,0,blend_radius_m)
    movel([0.129321, -1.314687, -2.613651, -0.784051, 1.570796, 1.700118],accel_mss,speed_ms,0,blend_radius_m)
    movel([0.128998, -1.314640, -2.613680, -0.784069, 1.570796, 1.699794],accel_mss,speed_ms,0,blend_radius_m)
    movel([0.128438, -1.314638, -2.613681, -0.784070, 1.570796, 1.699234],accel_mss,speed_ms,0,blend_radius_m)
    movel([0.128105, -1.314603, -2.613702, -0.784083, 1.570796, 1.698901],accel_mss,speed_ms,0,blend_radius_m)
    movel([0.127658, -1.314479, -2.613779, -0.784131, 1.570796, 1.698454],accel_mss,speed_ms,0,blend_radius_m)
    movel([0.127150, -1.314290, -2.613895, -0.784204, 1.570796, 1.697946],accel_mss,speed_ms,0,blend_radius_m)
    movel([0.126611, -1.314027, -2.614057, -0.784305, 1.570796, 1.697408],accel_mss,speed_ms,0,blend_radius_m)
    movel([0.126138, -1.313740, -2.614233, -0.784416, 1.570796, 1.696934],accel_mss,speed_ms,0,blend_radius_m)
    movel([0.126026, -1.313308, -2.614498, -0.784582, 1.570796, 1.696822],accel_mss,speed_ms,0,blend_radius_m)
    movel([0.125825, -1.313152, -2.614594, -0.784643, 1.570796, 1.696622],accel_mss,speed_ms,0,blend_radius_m)
    movel([0.125574, -1.313101, -2.614625, -0.784663, 1.570796, 1.696370],accel_mss,speed_ms,0,blend_radius_m)
    movel([0.125272, -1.313076, -2.614640, -0.784672, 1.570796, 1.696068],accel_mss,speed_ms,0,blend_radius_m)
    movel([0.125327, -1.312813, -2.614802, -0.784774, 1.570796, 1.696123],accel_mss,speed_ms,0,blend_radius_m)
    movel([0.126338, -1.312056, -2.615266, -0.785068, 1.570796, 1.697134],accel_mss,speed_ms,0,blend_radius_m)
    movel([0.126809, -1.311735, -2.615462, -0.785192, 1.570796, 1.697605],accel_mss,speed_ms,0,blend_radius_m)
    movel([0.127236, -1.311466, -2.615626, -0.785297, 1.570796, 1.698032],accel_mss,speed_ms,0,blend_radius_m)
    movel([0.127546, -1.311290, -2.615734, -0.785365, 1.570796, 1.698343],accel_mss,speed_ms,0,blend_radius_m)
    movel([0.127887, -1.311121, -2.615837, -0.785431, 1.570796, 1.698683],accel_mss,speed_ms,0,blend_radius_m)
    movel([0.128246, -1.310967, -2.615931, -0.785491, 1.570796, 1.699042],accel_mss,speed_ms,0,blend_radius_m)
    movel([0.128661, -1.310818, -2.616022, -0.785549, 1.570796, 1.699458],accel_mss,speed_ms,0,blend_radius_m)
    movel([0.129189, -1.310664, -2.616116, -0.785609, 1.570796, 1.699986],accel_mss,speed_ms,0,blend_radius_m)
    movel([0.129849, -1.310495, -2.616219, -0.785675, 1.570796, 1.700645],accel_mss,speed_ms,0,blend_radius_m)
    movel([0.130352, -1.310389, -2.616284, -0.785716, 1.570796, 1.701148],accel_mss,speed_ms,0,blend_radius_m)
    movel([0.130822, -1.310313, -2.616330, -0.785746, 1.570796, 1.701618],accel_mss,speed_ms,0,blend_radius_m)
    movel([0.131291, -1.310260, -2.616362, -0.785766, 1.570796, 1.702087],accel_mss,speed_ms,0,blend_radius_m)
    movel([0.131727, -1.310236, -2.616377, -0.785776, 1.570796, 1.702523],accel_mss,speed_ms,0,blend_radius_m)
    movel([0.132109, -1.310244, -2.616372, -0.785773, 1.570796, 1.702906],accel_mss,speed_ms,0,blend_radius_m)
    movel([0.132614, -1.310303, -2.616336, -0.785750, 1.570796, 1.703410],accel_mss,speed_ms,0,blend_radius_m)
    movel([0.133084, -1.310416, -2.616267, -0.785706, 1.570796, 1.703880],accel_mss,speed_ms,0,blend_radius_m)
    movel([0.133497, -1.310581, -2.616167, -0.785642, 1.570796, 1.704293],accel_mss,speed_ms,0,blend_radius_m)
    movel([0.133863, -1.310801, -2.616033, -0.785556, 1.570796, 1.704659],accel_mss,speed_ms,0,blend_radius_m)
    movel([0.134195, -1.311084, -2.615860, -0.785446, 1.570796, 1.704992],accel_mss,speed_ms,0,blend_radius_m)
    movel([0.134483, -1.311423, -2.615652, -0.785313, 1.570796, 1.705279],accel_mss,speed_ms,0,blend_radius_m)
    movel([0.134709, -1.311792, -2.615427, -0.785170, 1.570796, 1.705505],accel_mss,speed_ms,0,blend_radius_m)
    movel([0.134897, -1.312237, -2.615155, -0.784997, 1.570796, 1.705694],accel_mss,speed_ms,0,blend_radius_m)
    movel([0.135030, -1.312690, -2.614877, -0.784822, 1.570796, 1.705827],accel_mss,speed_ms,0,blend_radius_m)
    movel([0.135100, -1.313096, -2.614628, -0.784664, 1.570796, 1.705897],accel_mss,speed_ms,0,blend_radius_m)
    movel([0.135107, -1.313513, -2.614372, -0.784503, 1.570796, 1.705903],accel_mss,speed_ms,0,blend_radius_m)
    movel([0.135051, -1.313950, -2.614104, -0.784335, 1.570796, 1.705847],accel_mss,speed_ms,0,blend_radius_m)
    movel([0.134944, -1.314385, -2.613837, -0.784167, 1.570796, 1.705740],accel_mss,speed_ms,0,blend_radius_m)
    movel([0.134785, -1.314825, -2.613566, -0.783998, 1.570796, 1.705581],accel_mss,speed_ms,0,blend_radius_m)
    movel([0.134510, -1.315429, -2.613194, -0.783766, 1.570796, 1.705307],accel_mss,speed_ms,0,blend_radius_m)
    movel([0.134188, -1.316033, -2.612822, -0.783535, 1.570796, 1.704984],accel_mss,speed_ms,0,blend_radius_m)
    movel([0.134188, -1.318953, -2.614172, -0.779264, 1.570796, 1.704984],accel_mss,speed_ms,0,blend_radius_m)
    movel([0.133863, -1.319471, -2.613851, -0.779067, 1.570796, 1.704659],accel_mss,speed_ms,0,blend_radius_m)
    movel([0.133488, -1.319979, -2.613535, -0.778875, 1.570796, 1.704284],accel_mss,speed_ms,0,blend_radius_m)
    movel([0.133051, -1.320491, -2.613217, -0.778681, 1.570796, 1.703848],accel_mss,speed_ms,0,blend_radius_m)
    movel([0.132574, -1.320986, -2.612909, -0.778494, 1.570796, 1.703370],accel_mss,speed_ms,0,blend_radius_m)
    movel([0.132063, -1.321455, -2.612617, -0.778317, 1.570796, 1.702859],accel_mss,speed_ms,0,blend_radius_m)
    movel([0.131519, -1.321898, -2.612341, -0.778150, 1.570796, 1.702316],accel_mss,speed_ms,0,blend_radius_m)
    movel([0.130956, -1.322305, -2.612087, -0.777997, 1.570796, 1.701752],accel_mss,speed_ms,0,blend_radius_m)
    movel([0.130359, -1.322685, -2.611849, -0.777854, 1.570796, 1.701155],accel_mss,speed_ms,0,blend_radius_m)
    movel([0.129758, -1.323021, -2.611639, -0.777728, 1.570796, 1.700554],accel_mss,speed_ms,0,blend_radius_m)
    movel([0.129170, -1.323305, -2.611462, -0.777622, 1.570796, 1.699967],accel_mss,speed_ms,0,blend_radius_m)
    movel([0.128584, -1.323546, -2.611311, -0.777532, 1.570796, 1.699380],accel_mss,speed_ms,0,blend_radius_m)
    movel([0.127997, -1.323736, -2.611192, -0.777461, 1.570796, 1.698794],accel_mss,speed_ms,0,blend_radius_m)
    movel([0.127420, -1.323881, -2.611101, -0.777407, 1.570796, 1.698216],accel_mss,speed_ms,0,blend_radius_m)
    movel([0.126855, -1.323975, -2.611043, -0.777372, 1.570796, 1.697652],accel_mss,speed_ms,0,blend_radius_m)
    movel([0.126287, -1.324019, -2.611015, -0.777355, 1.570796, 1.697084],accel_mss,speed_ms,0,blend_radius_m)
    movel([0.125741, -1.324017, -2.611016, -0.777356, 1.570796, 1.696538],accel_mss,speed_ms,0,blend_radius_m)
    movel([0.125218, -1.323962, -2.611050, -0.777376, 1.570796, 1.696014],accel_mss,speed_ms,0,blend_radius_m)
    movel([0.124728, -1.323855, -2.611118, -0.777416, 1.570796, 1.695524],accel_mss,speed_ms,0,blend_radius_m)
    movel([0.124274, -1.323703, -2.611213, -0.777473, 1.570796, 1.695070],accel_mss,speed_ms,0,blend_radius_m)
    movel([0.123865, -1.323505, -2.611337, -0.777547, 1.570796, 1.694662],accel_mss,speed_ms,0,blend_radius_m)
    movel([0.123500, -1.323255, -2.611493, -0.777641, 1.570796, 1.694296],accel_mss,speed_ms,0,blend_radius_m)
    movel([0.123179, -1.322960, -2.611678, -0.777751, 1.570796, 1.693975],accel_mss,speed_ms,0,blend_radius_m)
    movel([0.122903, -1.322615, -2.611893, -0.777881, 1.570796, 1.693699],accel_mss,speed_ms,0,blend_radius_m)
    movel([0.122698, -1.322254, -2.612118, -0.778016, 1.570796, 1.693494],accel_mss,speed_ms,0,blend_radius_m)
    movel([0.122566, -1.321888, -2.612347, -0.778154, 1.570796, 1.693362],accel_mss,speed_ms,0,blend_radius_m)
    movel([0.122485, -1.321491, -2.612594, -0.778303, 1.570796, 1.693281],accel_mss,speed_ms,0,blend_radius_m)
    movel([0.122458, -1.321069, -2.612858, -0.778463, 1.570796, 1.693255],accel_mss,speed_ms,0,blend_radius_m)
    movel([0.122486, -1.320625, -2.613134, -0.778630, 1.570796, 1.693283],accel_mss,speed_ms,0,blend_radius_m)
    movel([0.122590, -1.320024, -2.613507, -0.778858, 1.570796, 1.693386],accel_mss,speed_ms,0,blend_radius_m)
    movel([0.122748, -1.319407, -2.613891, -0.779092, 1.570796, 1.693544],accel_mss,speed_ms,0,blend_radius_m)
    movel([0.122933, -1.318870, -2.614223, -0.779296, 1.570796, 1.693730],accel_mss,speed_ms,0,blend_radius_m)
    movel([0.123172, -1.318341, -2.614551, -0.779497, 1.570796, 1.693969],accel_mss,speed_ms,0,blend_radius_m)
    movel([0.123393, -1.317942, -2.614798, -0.779649, 1.570796, 1.694190],accel_mss,speed_ms,0,blend_radius_m)
    movel([0.123730, -1.317588, -2.615016, -0.779784, 1.570796, 1.694526],accel_mss,speed_ms,0,blend_radius_m)
    movel([0.124098, -1.317451, -2.615102, -0.779837, 1.570796, 1.694894],accel_mss,speed_ms,0,blend_radius_m)
    movel([0.124241, -1.317611, -2.615002, -0.779775, 1.570796, 1.695037],accel_mss,speed_ms,0,blend_radius_m)
    movel([0.124444, -1.317750, -2.614917, -0.779723, 1.570796, 1.695240],accel_mss,speed_ms,0,blend_radius_m)
    movel([0.125111, -1.317746, -2.614919, -0.779724, 1.570796, 1.695907],accel_mss,speed_ms,0,blend_radius_m)
    movel([0.125436, -1.317782, -2.614897, -0.779710, 1.570796, 1.696233],accel_mss,speed_ms,0,blend_radius_m)
    movel([0.125718, -1.317873, -2.614841, -0.779676, 1.570796, 1.696514],accel_mss,speed_ms,0,blend_radius_m)
    movel([0.126039, -1.317993, -2.614766, -0.779630, 1.570796, 1.696836],accel_mss,speed_ms,0,blend_radius_m)
    movel([0.126622, -1.318272, -2.614593, -0.779523, 1.570796, 1.697418],accel_mss,speed_ms,0,blend_radius_m)
    movel([0.127045, -1.318524, -2.614437, -0.779427, 1.570796, 1.697841],accel_mss,speed_ms,0,blend_radius_m)
    movel([0.127393, -1.318780, -2.614279, -0.779330, 1.570796, 1.698189],accel_mss,speed_ms,0,blend_radius_m)
    movel([0.127590, -1.319006, -2.614139, -0.779244, 1.570796, 1.698386],accel_mss,speed_ms,0,blend_radius_m)
    movel([0.127760, -1.319308, -2.613952, -0.779129, 1.570796, 1.698556],accel_mss,speed_ms,0,blend_radius_m)
    movel([0.127974, -1.319543, -2.613806, -0.779040, 1.570796, 1.698770],accel_mss,speed_ms,0,blend_radius_m)
    movel([0.128319, -1.319682, -2.613720, -0.778987, 1.570796, 1.699116],accel_mss,speed_ms,0,blend_radius_m)
    movel([0.128768, -1.319621, -2.613757, -0.779010, 1.570796, 1.699565],accel_mss,speed_ms,0,blend_radius_m)
    movel([0.129117, -1.319438, -2.613871, -0.779080, 1.570796, 1.699913],accel_mss,speed_ms,0,blend_radius_m)
    movel([0.129483, -1.319115, -2.614072, -0.779203, 1.570796, 1.700280],accel_mss,speed_ms,0,blend_radius_m)
    movel([0.129679, -1.318868, -2.614225, -0.779297, 1.570796, 1.700476],accel_mss,speed_ms,0,blend_radius_m)
    movel([0.129887, -1.318383, -2.614525, -0.779481, 1.570796, 1.700683],accel_mss,speed_ms,0,blend_radius_m)
    movel([0.129841, -1.317972, -2.614779, -0.779638, 1.570796, 1.700637],accel_mss,speed_ms,0,blend_radius_m)
    movel([0.129723, -1.317813, -2.614878, -0.779698, 1.570796, 1.700519],accel_mss,speed_ms,0,blend_radius_m)
    movel([0.129545, -1.317689, -2.614954, -0.779746, 1.570796, 1.700341],accel_mss,speed_ms,0,blend_radius_m)
    movel([0.129321, -1.317611, -2.615003, -0.779776, 1.570796, 1.700118],accel_mss,speed_ms,0,blend_radius_m)
    movel([0.128998, -1.317564, -2.615032, -0.779794, 1.570796, 1.699794],accel_mss,speed_ms,0,blend_radius_m)
    movel([0.128438, -1.317562, -2.615033, -0.779794, 1.570796, 1.699234],accel_mss,speed_ms,0,blend_radius_m)
    movel([0.128105, -1.317527, -2.615054, -0.779808, 1.570796, 1.698901],accel_mss,speed_ms,0,blend_radius_m)
    movel([0.127658, -1.317403, -2.615131, -0.779855, 1.570796, 1.698454],accel_mss,speed_ms,0,blend_radius_m)
    movel([0.127150, -1.317214, -2.615248, -0.779927, 1.570796, 1.697946],accel_mss,speed_ms,0,blend_radius_m)
    movel([0.126611, -1.316952, -2.615410, -0.780028, 1.570796, 1.697408],accel_mss,speed_ms,0,blend_radius_m)
    movel([0.126138, -1.316665, -2.615586, -0.780137, 1.570796, 1.696934],accel_mss,speed_ms,0,blend_radius_m)
    movel([0.126026, -1.316235, -2.615852, -0.780303, 1.570796, 1.696822],accel_mss,speed_ms,0,blend_radius_m)
    movel([0.125825, -1.316079, -2.615948, -0.780362, 1.570796, 1.696622],accel_mss,speed_ms,0,blend_radius_m)
    movel([0.125574, -1.316028, -2.615979, -0.780382, 1.570796, 1.696370],accel_mss,speed_ms,0,blend_radius_m)
    movel([0.125272, -1.316003, -2.615995, -0.780391, 1.570796, 1.696068],accel_mss,speed_ms,0,blend_radius_m)
    movel([0.125327, -1.315740, -2.616157, -0.780493, 1.570796, 1.696123],accel_mss,speed_ms,0,blend_radius_m)
    movel([0.126338, -1.314984, -2.616621, -0.780783, 1.570796, 1.697134],accel_mss,speed_ms,0,blend_radius_m)
    movel([0.126809, -1.314664, -2.616818, -0.780907, 1.570796, 1.697605],accel_mss,speed_ms,0,blend_radius_m)
    movel([0.127236, -1.314396, -2.616982, -0.781010, 1.570796, 1.698032],accel_mss,speed_ms,0,blend_radius_m)
    movel([0.127546, -1.314220, -2.617091, -0.781078, 1.570796, 1.698343],accel_mss,speed_ms,0,blend_radius_m)
    movel([0.127887, -1.314051, -2.617194, -0.781144, 1.570796, 1.698683],accel_mss,speed_ms,0,blend_radius_m)
    movel([0.128246, -1.313898, -2.617288, -0.781203, 1.570796, 1.699042],accel_mss,speed_ms,0,blend_radius_m)
    movel([0.128661, -1.313749, -2.617379, -0.781261, 1.570796, 1.699458],accel_mss,speed_ms,0,blend_radius_m)
    movel([0.129189, -1.313596, -2.617473, -0.781320, 1.570796, 1.699986],accel_mss,speed_ms,0,blend_radius_m)
    movel([0.129849, -1.313427, -2.617576, -0.781385, 1.570796, 1.700645],accel_mss,speed_ms,0,blend_radius_m)
    movel([0.130352, -1.313321, -2.617642, -0.781427, 1.570796, 1.701148],accel_mss,speed_ms,0,blend_radius_m)
    movel([0.130822, -1.313245, -2.617688, -0.781456, 1.570796, 1.701618],accel_mss,speed_ms,0,blend_radius_m)
    movel([0.131291, -1.313193, -2.617720, -0.781476, 1.570796, 1.702087],accel_mss,speed_ms,0,blend_radius_m)
    movel([0.131727, -1.313169, -2.617735, -0.781486, 1.570796, 1.702523],accel_mss,speed_ms,0,blend_radius_m)
    movel([0.132109, -1.313176, -2.617730, -0.781482, 1.570796, 1.702906],accel_mss,speed_ms,0,blend_radius_m)
    movel([0.132614, -1.313235, -2.617694, -0.781460, 1.570796, 1.703410],accel_mss,speed_ms,0,blend_radius_m)
    movel([0.133084, -1.313348, -2.617625, -0.781416, 1.570796, 1.703880],accel_mss,speed_ms,0,blend_radius_m)
    movel([0.133497, -1.313512, -2.617524, -0.781352, 1.570796, 1.704293],accel_mss,speed_ms,0,blend_radius_m)
    movel([0.133863, -1.313732, -2.617390, -0.781267, 1.570796, 1.704659],accel_mss,speed_ms,0,blend_radius_m)
    movel([0.134195, -1.314014, -2.617217, -0.781158, 1.570796, 1.704992],accel_mss,speed_ms,0,blend_radius_m)
    movel([0.134483, -1.314353, -2.617009, -0.781027, 1.570796, 1.705279],accel_mss,speed_ms,0,blend_radius_m)
    movel([0.134709, -1.314722, -2.616783, -0.780885, 1.570796, 1.705505],accel_mss,speed_ms,0,blend_radius_m)
    movel([0.134897, -1.315165, -2.616510, -0.780714, 1.570796, 1.705694],accel_mss,speed_ms,0,blend_radius_m)
    movel([0.135030, -1.315618, -2.616232, -0.780540, 1.570796, 1.705827],accel_mss,speed_ms,0,blend_radius_m)
    movel([0.135100, -1.316023, -2.615982, -0.780384, 1.570796, 1.705897],accel_mss,speed_ms,0,blend_radius_m)
    movel([0.135107, -1.316439, -2.615726, -0.780224, 1.570796, 1.705903],accel_mss,speed_ms,0,blend_radius_m)
    movel([0.135051, -1.316875, -2.615457, -0.780057, 1.570796, 1.705847],accel_mss,speed_ms,0,blend_radius_m)
    movel([0.134944, -1.317309, -2.615189, -0.779891, 1.570796, 1.705740],accel_mss,speed_ms,0,blend_radius_m)
    movel([0.134785, -1.317748, -2.614918, -0.779723, 1.570796, 1.705581],accel_mss,speed_ms,0,blend_radius_m)
    movel([0.134510, -1.318351, -2.614545, -0.779493, 1.570796, 1.705307],accel_mss,speed_ms,0,blend_radius_m)
    movel([0.134188, -1.318953, -2.614172, -0.779264, 1.570796, 1.704984],accel_mss,speed_ms,0,blend_radius_m)
    movel([0.134188, -1.285153, -2.597586, -0.829650, 1.570796, 1.704984],accel_mss,speed_ms,0,blend_radius_m)
    speed_ms = 1.000
    movel([0.137251, -1.275756, -2.603080, -0.833553, 1.570796, 1.708047],accel_mss,speed_ms,0,blend_radius_m)
    speed_ms = 0.008
    movel([0.137251, -1.303314, -2.616821, -0.792254, 1.570796, 1.708047],accel_mss,speed_ms,0,blend_radius_m)
    speed_ms = 0.003
    movel([0.137251, -1.306806, -2.618460, -0.787123, 1.570796, 1.708047],accel_mss,speed_ms,0,blend_radius_m)
    speed_ms = 0.008
    movel([0.136956, -1.306799, -2.618464, -0.787126, 1.570796, 1.707752],accel_mss,speed_ms,0,blend_radius_m)
    movel([0.136646, -1.306820, -2.618451, -0.787118, 1.570796, 1.707442],accel_mss,speed_ms,0,blend_radius_m)
    movel([0.136330, -1.306867, -2.618423, -0.787099, 1.570796, 1.707126],accel_mss,speed_ms,0,blend_radius_m)
    movel([0.136004, -1.306941, -2.618378, -0.787070, 1.570796, 1.706800],accel_mss,speed_ms,0,blend_radius_m)
    movel([0.130263, -1.308634, -2.617352, -0.786403, 1.570796, 1.701060],accel_mss,speed_ms,0,blend_radius_m)
    movel([0.122240, -1.311092, -2.615855, -0.785442, 1.570796, 1.693036],accel_mss,speed_ms,0,blend_radius_m)
    movel([0.121881, -1.311266, -2.615749, -0.785375, 1.570796, 1.692677],accel_mss,speed_ms,0,blend_radius_m)
    movel([0.121557, -1.311529, -2.615588, -0.785272, 1.570796, 1.692353],accel_mss,speed_ms,0,blend_radius_m)
    movel([0.121274, -1.311902, -2.615360, -0.785127, 1.570796, 1.692071],accel_mss,speed_ms,0,blend_radius_m)
    movel([0.121125, -1.312291, -2.615121, -0.784976, 1.570796, 1.691922],accel_mss,speed_ms,0,blend_radius_m)
    movel([0.120597, -1.315805, -2.612962, -0.783622, 1.570796, 1.691393],accel_mss,speed_ms,0,blend_radius_m)
    movel([0.120081, -1.319359, -2.610762, -0.782268, 1.570796, 1.690877],accel_mss,speed_ms,0,blend_radius_m)
    movel([0.119488, -1.323654, -2.608080, -0.780655, 1.570796, 1.690285],accel_mss,speed_ms,0,blend_radius_m)
    movel([0.119491, -1.323881, -2.607937, -0.780571, 1.570796, 1.690287],accel_mss,speed_ms,0,blend_radius_m)
